LIN {X 0,Y 736.323,Z 990.485,A -85,B 0,C 180,E1 33731.391,E2 33731.391} C_VEL
LIN {X 0,Y 736.504,Z 974.64,A -85,B 0,C 180,E1 33729.663,E2 33729.663} C_VEL
LIN {X 0,Y 736.684,Z 957.169,A -85,B 0,C 180,E1 33728,E2 33728} C_VEL
LIN {X 0,Y 736.943,Z 939.859,A -85,B 0,C 180,E1 33726.521,E2 33726.521} C_VEL
LIN {X 0,Y 737.195,Z 919.804,A -85,B 0,C 180,E1 33725.008,E2 33725.008} C_VEL
LIN {X 0,Y 737.439,Z 901.418,A -85,B 0,C 180,E1 33723.767,E2 33723.767} C_VEL
LIN {X 0,Y 737.809,Z 878.245,A -85,B 0,C 180,E1 33722.388,E2 33722.388} C_VEL
LIN {X 0,Y 738.071,Z 858.185,A -85,B 0,C 180,E1 33721.343,E2 33721.343} C_VEL
LIN {X 0,Y 738.362,Z 837.251,A -85,B 0,C 180,E1 33720.378,E2 33720.378} C_VEL
LIN {X 0,Y 738.709,Z 812.608,A -85,B 0,C 180,E1 33719.407,E2 33719.407} C_VEL
LIN {X 0,Y 738.944,Z 791.175,A -85,B 0,C 180,E1 33718.695,E2 33718.695} C_VEL
LIN {X 0,Y 739.147,Z 770.122,A -85,B 0,C 180,E1 33718.104,E2 33718.104} C_VEL
LIN {X 0,Y 739.421,Z 744.677,A -85,B 0,C 180,E1 33717.531,E2 33717.531} C_VEL
LIN {X 0,Y 739.56,Z 720.624,A -85,B 0,C 180,E1 33717.14,E2 33717.14} C_VEL
LIN {X 0,Y 739.828,Z 623.646,A -85,B 0,C 180,E1 33716.024,E2 33716.024} C_VEL
LIN {X 0,Y 740.398,Z 398.303,A -85,B 0,C 180,E1 33713.431,E2 33713.431} C_VEL
LIN {X 0,Y 740.567,Z 293.06,A -85,B 0,C 180,E1 33712.186,E2 33712.186} C_VEL
LIN {X 0,Y 739.192,Z 287.411,A -85,B 0,C 180,E1 33712.014,E2 33712.014} C_VEL
LIN {X 0,Y 739.245,Z 262.741,A -85,B 0,C 180,E1 33710.326,E2 33710.326} C_VEL
LIN {X 0,Y 736.098,Z 254.481,A -85,B 0,C 180,E1 33709.508,E2 33709.508} C_VEL
LIN {X 0,Y 736.036,Z 254.289,A -85,B 0,C 180,E1 33706.505,E2 33706.505} C_VEL
LIN {X 0,Y 736.021,Z 254.293,A -85,B 0,C 180,E1 33704.057,E2 33704.057} C_VEL
LIN {X 0,Y 736.063,Z 254.286,A -85,B 0,C 180,E1 33701.419,E2 33701.419} C_VEL
LIN {X 0,Y 736.038,Z 254.29,A -85,B 0,C 180,E1 33698.387,E2 33698.387} C_VEL
LIN {X 0,Y 736.02,Z 254.291,A -85,B 0,C 180,E1 33695.936,E2 33695.936} C_VEL
LIN {X 0,Y 736.055,Z 254.282,A -85,B 0,C 180,E1 33693.339,E2 33693.339} C_VEL
LIN {X 0,Y 736.049,Z 254.29,A -85,B 0,C 180,E1 33690.354,E2 33690.354} C_VEL
LIN {X 0,Y 736.019,Z 254.287,A -85,B 0,C 180,E1 33687.824,E2 33687.824} C_VEL
LIN {X 0,Y 736.05,Z 254.289,A -85,B 0,C 180,E1 33685.249,E2 33685.249} C_VEL
LIN {X 0,Y 736.045,Z 254.293,A -85,B 0,C 180,E1 33682.188,E2 33682.188} C_VEL
LIN {X 0,Y 736.018,Z 254.29,A -85,B 0,C 180,E1 33679.689,E2 33679.689} C_VEL
LIN {X 0,Y 736.047,Z 254.288,A -85,B 0,C 180,E1 33677.145,E2 33677.145} C_VEL
LIN {X 0,Y 736.047,Z 254.292,A -85,B 0,C 180,E1 33674.073,E2 33674.073} C_VEL
LIN {X 0,Y 736.019,Z 254.29,A -85,B 0,C 180,E1 33671.52,E2 33671.52} C_VEL
LIN {X 0,Y 736.058,Z 254.288,A -85,B 0,C 180,E1 33668.909,E2 33668.909} C_VEL
LIN {X 0,Y 736.045,Z 254.292,A -85,B 0,C 180,E1 33665.926,E2 33665.926} C_VEL
LIN {X 0,Y 736.018,Z 254.29,A -85,B 0,C 180,E1 33663.427,E2 33663.427} C_VEL
LIN {X 0,Y 736.04,Z 254.289,A -85,B 0,C 180,E1 33660.934,E2 33660.934} C_VEL
LIN {X 0,Y 736.057,Z 254.293,A -85,B 0,C 180,E1 33657.898,E2 33657.898} C_VEL
LIN {X 0,Y 736.018,Z 254.289,A -85,B 0,C 180,E1 33655.325,E2 33655.325} C_VEL
LIN {X 0,Y 736.037,Z 254.289,A -85,B 0,C 180,E1 33652.82,E2 33652.82} C_VEL
LIN {X 0,Y 736.066,Z 254.294,A -85,B 0,C 180,E1 33649.828,E2 33649.828} C_VEL
LIN {X 0,Y 736.017,Z 254.291,A -85,B 0,C 180,E1 33649.201,E2 33649.201} C_VEL
LIN {X 0,Y 735.014,Z 254.419,A -85,B 0,C 180,E1 33648.601,E2 33648.601} C_VEL
LIN {X 0,Y 728.702,Z 255.201,A -85,B 0,C 180,E1 33646.965,E2 33646.965} C_VEL
LIN {X 0,Y 728.126,Z 255.274,A -85,B 0,C 180,E1 33646.485,E2 33646.485} C_VEL
LIN {X 0,Y 728.097,Z 255.278,A -85,B 0,C 180,E1 33643.485,E2 33643.485} C_VEL
LIN {X 0,Y 728.079,Z 255.28,A -85,B 0,C 180,E1 33641.005,E2 33641.005} C_VEL
LIN {X 0,Y 728.121,Z 255.275,A -85,B 0,C 180,E1 33638.385,E2 33638.385} C_VEL
LIN {X 0,Y 728.1,Z 255.276,A -85,B 0,C 180,E1 33635.383,E2 33635.383} C_VEL
LIN {X 0,Y 728.078,Z 255.271,A -85,B 0,C 180,E1 33632.862,E2 33632.862} C_VEL
LIN {X 0,Y 728.117,Z 255.278,A -85,B 0,C 180,E1 33630.281,E2 33630.281} C_VEL
LIN {X 0,Y 728.098,Z 255.27,A -85,B 0,C 180,E1 33627.243,E2 33627.243} C_VEL
LIN {X 0,Y 728.078,Z 255.28,A -85,B 0,C 180,E1 33624.774,E2 33624.774} C_VEL
LIN {X 0,Y 728.106,Z 255.276,A -85,B 0,C 180,E1 33622.231,E2 33622.231} C_VEL
LIN {X 0,Y 728.106,Z 255.281,A -85,B 0,C 180,E1 33619.171,E2 33619.171} C_VEL
LIN {X 0,Y 728.078,Z 255.28,A -85,B 0,C 180,E1 33616.593,E2 33616.593} C_VEL
LIN {X 0,Y 728.121,Z 255.28,A -85,B 0,C 180,E1 33613.98,E2 33613.98} C_VEL
LIN {X 0,Y 728.096,Z 255.277,A -85,B 0,C 180,E1 33610.947,E2 33610.947} C_VEL
LIN {X 0,Y 728.077,Z 255.28,A -85,B 0,C 180,E1 33608.471,E2 33608.471} C_VEL
LIN {X 0,Y 728.174,Z 255.513,A -85,B 0,C 180,E1 33607.228,E2 33607.228} C_VEL
LIN {X 0,Y 732.4,Z 266.408,A -85,B 0,C 180,E1 33606.141,E2 33606.141} C_VEL
LIN {X 0,Y 732.336,Z 278.075,A -85,B 0,C 180,E1 33605.34,E2 33605.34} C_VEL
LIN {X 0,Y 734.39,Z 286.67,A -85,B 0,C 180,E1 33605.1,E2 33605.1} C_VEL
LIN {X 0,Y 733.457,Z 536.818,A -85,B 0,C 180,E1 33602.164,E2 33602.164} C_VEL
LIN {X 0,Y 732.828,Z 710.294,A -85,B 0,C 180,E1 33600.161,E2 33600.161} C_VEL
LIN {X 0,Y 732.643,Z 734.058,A -85,B 0,C 180,E1 33599.773,E2 33599.773} C_VEL
LIN {X 0,Y 732.274,Z 759.946,A -85,B 0,C 180,E1 33599.191,E2 33599.191} C_VEL
LIN {X 0,Y 731.999,Z 780.748,A -85,B 0,C 180,E1 33598.605,E2 33598.605} C_VEL
LIN {X 0,Y 731.681,Z 802.912,A -85,B 0,C 180,E1 33597.863,E2 33597.863} C_VEL
LIN {X 0,Y 731.192,Z 828.846,A -85,B 0,C 180,E1 33596.825,E2 33596.825} C_VEL
LIN {X 0,Y 730.818,Z 849.11,A -85,B 0,C 180,E1 33595.877,E2 33595.877} C_VEL
LIN {X 0,Y 730.44,Z 871.706,A -85,B 0,C 180,E1 33594.677,E2 33594.677} C_VEL
LIN {X 0,Y 729.958,Z 893.15,A -85,B 0,C 180,E1 33593.363,E2 33593.363} C_VEL
LIN {X 0,Y 729.63,Z 912.174,A -85,B 0,C 180,E1 33592.054,E2 33592.054} C_VEL
LIN {X 0,Y 729.24,Z 932.601,A -85,B 0,C 180,E1 33590.465,E2 33590.465} C_VEL
LIN {X 0,Y 728.948,Z 948.78,A -85,B 0,C 180,E1 33589.054,E2 33589.054} C_VEL
LIN {X 0,Y 728.657,Z 967.272,A -85,B 0,C 180,E1 33587.238,E2 33587.238} C_VEL
LIN {X 0,Y 728.462,Z 981.209,A -85,B 0,C 180,E1 33585.688,E2 33585.688} C_VEL
LIN {X 0,Y 728.285,Z 995.564,A -85,B 0,C 180,E1 33583.902,E2 33583.902} C_VEL
LIN {X 0,Y 728.133,Z 1008.414,A -85,B 0,C 180,E1 33582.048,E2 33582.048} C_VEL
LIN {X 0,Y 728.063,Z 1018.17,A -85,B 0,C 180,E1 33580.444,E2 33580.444} C_VEL
LIN {X 0,Y 727.999,Z 1027.486,A -85,B 0,C 180,E1 33578.69,E2 33578.69} C_VEL
LIN {X 0,Y 727.93,Z 1036.565,A -85,B 0,C 180,E1 33576.626,E2 33576.626} C_VEL
LIN {X 0,Y 727.926,Z 1042.525,A -85,B 0,C 180,E1 33574.964,E2 33574.964} C_VEL
LIN {X 0,Y 727.917,Z 1047.127,A -85,B 0,C 180,E1 33573.386,E2 33573.386} C_VEL
LIN {X 0,Y 727.895,Z 1051.021,A -85,B 0,C 180,E1 33571.653,E2 33571.653} C_VEL
LIN {X 0,Y 727.915,Z 1054.124,A -85,B 0,C 180,E1 33569.528,E2 33569.528} C_VEL
LIN {X 0,Y 727.898,Z 1055.29,A -85,B 0,C 180,E1 33567.717,E2 33567.717} C_VEL
LIN {X 0,Y 727.906,Z 1055.253,A -85,B 0,C 180,E1 33566.062,E2 33566.062} C_VEL
LIN {X 0,Y 727.915,Z 1053.741,A -85,B 0,C 180,E1 33563.998,E2 33563.998} C_VEL
LIN {X 0,Y 727.903,Z 1050.624,A -85,B 0,C 180,E1 33562.06,E2 33562.06} C_VEL
LIN {X 0,Y 727.919,Z 1046.681,A -85,B 0,C 180,E1 33560.353,E2 33560.353} C_VEL
LIN {X 0,Y 727.922,Z 1041.132,A -85,B 0,C 180,E1 33558.511,E2 33558.511} C_VEL
LIN {X 0,Y 727.968,Z 1033.315,A -85,B 0,C 180,E1 33556.497,E2 33556.497} C_VEL
LIN {X 0,Y 728.01,Z 1025.304,A -85,B 0,C 180,E1 33554.792,E2 33554.792} C_VEL
LIN {X 0,Y 728.07,Z 1016.391,A -85,B 0,C 180,E1 33553.156,E2 33553.156} C_VEL
LIN {X 0,Y 728.192,Z 1003.884,A -85,B 0,C 180,E1 33551.175,E2 33551.175} C_VEL
LIN {X 0,Y 728.339,Z 991.104,A -85,B 0,C 180,E1 33549.436,E2 33549.436} C_VEL
LIN {X 0,Y 728.522,Z 977.09,A -85,B 0,C 180,E1 33547.74,E2 33547.74} C_VEL
LIN {X 0,Y 728.764,Z 960.225,A -85,B 0,C 180,E1 33545.953,E2 33545.953} C_VEL
LIN {X 0,Y 729.023,Z 944.707,A -85,B 0,C 180,E1 33544.486,E2 33544.486} C_VEL
LIN {X 0,Y 729.396,Z 923.992,A -85,B 0,C 180,E1 33542.751,E2 33542.751} C_VEL
LIN {X 0,Y 729.722,Z 906.229,A -85,B 0,C 180,E1 33541.432,E2 33541.432} C_VEL
LIN {X 0,Y 730.18,Z 884.008,A -85,B 0,C 180,E1 33539.967,E2 33539.967} C_VEL
LIN {X 0,Y 730.522,Z 864.046,A -85,B 0,C 180,E1 33538.811,E2 33538.811} C_VEL
LIN {X 0,Y 730.942,Z 843.542,A -85,B 0,C 180,E1 33537.758,E2 33537.758} C_VEL
LIN {X 0,Y 731.406,Z 818.409,A -85,B 0,C 180,E1 33536.646,E2 33536.646} C_VEL
LIN {X 0,Y 731.725,Z 797.529,A -85,B 0,C 180,E1 33535.856,E2 33535.856} C_VEL
LIN {X 0,Y 732.078,Z 775.308,A -85,B 0,C 180,E1 33535.139,E2 33535.139} C_VEL
LIN {X 0,Y 732.452,Z 749.2,A -85,B 0,C 180,E1 33534.46,E2 33534.46} C_VEL
LIN {X 0,Y 732.673,Z 727.248,A -85,B 0,C 180,E1 33534.016,E2 33534.016} C_VEL
LIN {X 0,Y 732.842,Z 706.664,A -85,B 0,C 180,E1 33533.701,E2 33533.701} C_VEL
LIN {X 0,Y 733.756,Z 454.635,A -85,B 0,C 180,E1 33530.792,E2 33530.792} C_VEL
LIN {X 0,Y 734.238,Z 285.309,A -85,B 0,C 180,E1 33528.784,E2 33528.784} C_VEL
LIN {X 0,Y 732.302,Z 277.803,A -85,B 0,C 180,E1 33528.557,E2 33528.557} C_VEL
LIN {X 0,Y 732.281,Z 266.077,A -85,B 0,C 180,E1 33527.738,E2 33527.738} C_VEL
LIN {X 0,Y 728.187,Z 255.602,A -85,B 0,C 180,E1 33526.699,E2 33526.699} C_VEL
LIN {X 0,Y 728.128,Z 255.249,A -85,B 0,C 180,E1 33526.094,E2 33526.094} C_VEL
LIN {X 0,Y 728.079,Z 255.278,A -85,B 0,C 180,E1 33523.475,E2 33523.475} C_VEL
LIN {X 0,Y 728.096,Z 255.285,A -85,B 0,C 180,E1 33520.948,E2 33520.948} C_VEL
LIN {X 0,Y 728.132,Z 255.273,A -85,B 0,C 180,E1 33517.967,E2 33517.967} C_VEL
LIN {X 0,Y 728.08,Z 255.281,A -85,B 0,C 180,E1 33515.322,E2 33515.322} C_VEL
LIN {X 0,Y 728.095,Z 255.281,A -85,B 0,C 180,E1 33512.812,E2 33512.812} C_VEL
LIN {X 0,Y 728.127,Z 255.277,A -85,B 0,C 180,E1 33509.787,E2 33509.787} C_VEL
LIN {X 0,Y 728.079,Z 255.279,A -85,B 0,C 180,E1 33507.138,E2 33507.138} C_VEL
LIN {X 0,Y 728.103,Z 255.275,A -85,B 0,C 180,E1 33504.589,E2 33504.589} C_VEL
LIN {X 0,Y 728.109,Z 255.274,A -85,B 0,C 180,E1 33501.51,E2 33501.51} C_VEL
LIN {X 0,Y 728.079,Z 255.274,A -85,B 0,C 180,E1 33498.995,E2 33498.995} C_VEL
LIN {X 0,Y 728.107,Z 255.283,A -85,B 0,C 180,E1 33496.433,E2 33496.433} C_VEL
LIN {X 0,Y 728.103,Z 255.27,A -85,B 0,C 180,E1 33493.339,E2 33493.339} C_VEL
LIN {X 0,Y 728.08,Z 255.28,A -85,B 0,C 180,E1 33490.845,E2 33490.845} C_VEL
LIN {X 0,Y 728.108,Z 255.28,A -85,B 0,C 180,E1 33488.291,E2 33488.291} C_VEL
LIN {X 0,Y 728.104,Z 255.276,A -85,B 0,C 180,E1 33485.2,E2 33485.2} C_VEL
LIN {X 0,Y 728.079,Z 255.28,A -85,B 0,C 180,E1 33482.676,E2 33482.676} C_VEL
LIN {X 0,Y 728.117,Z 255.274,A -85,B 0,C 180,E1 33480.079,E2 33480.079} C_VEL
LIN {X 0,Y 728.099,Z 255.279,A -85,B 0,C 180,E1 33477.009,E2 33477.009} C_VEL
LIN {X 0,Y 728.08,Z 255.277,A -85,B 0,C 180,E1 33474.483,E2 33474.483} C_VEL
LIN {X 0,Y 728.14,Z 255.272,A -85,B 0,C 180,E1 33471.789,E2 33471.789} C_VEL
LIN {X 0,Y 728.095,Z 255.277,A -85,B 0,C 180,E1 33468.835,E2 33468.835} C_VEL
LIN {X 0,Y 728.08,Z 255.27,A -85,B 0,C 180,E1 33466.337,E2 33466.337} C_VEL
LIN {X 0,Y 728.141,Z 255.28,A -85,B 0,C 180,E1 33463.65,E2 33463.65} C_VEL
LIN {X 0,Y 728.094,Z 255.271,A -85,B 0,C 180,E1 33460.673,E2 33460.673} C_VEL
LIN {X 0,Y 728.082,Z 255.277,A -85,B 0,C 180,E1 33458.18,E2 33458.18} C_VEL
LIN {X 0,Y 728.145,Z 255.283,A -85,B 0,C 180,E1 33455.499,E2 33455.499} C_VEL
LIN {X 0,Y 728.093,Z 255.278,A -85,B 0,C 180,E1 33452.517,E2 33452.517} C_VEL
LIN {X 0,Y 728.082,Z 255.281,A -85,B 0,C 180,E1 33450.061,E2 33450.061} C_VEL
LIN {X 0,Y 728.147,Z 255.271,A -85,B 0,C 180,E1 33447.327,E2 33447.327} C_VEL
LIN {X 0,Y 728.093,Z 255.28,A -85,B 0,C 180,E1 33444.389,E2 33444.389} C_VEL
LIN {X 0,Y 728.083,Z 255.271,A -85,B 0,C 180,E1 33441.897,E2 33441.897} C_VEL
LIN {X 0,Y 728.154,Z 255.282,A -85,B 0,C 180,E1 33439.167,E2 33439.167} C_VEL
LIN {X 0,Y 728.093,Z 255.28,A -85,B 0,C 180,E1 33436.249,E2 33436.249} C_VEL
LIN {X 0,Y 728.082,Z 255.276,A -85,B 0,C 180,E1 33433.749,E2 33433.749} C_VEL
LIN {X 0,Y 728.193,Z 255.483,A -85,B 0,C 180,E1 33430.95,E2 33430.95} C_VEL
LIN {X 0,Y 732.603,Z 267.238,A -85,B 0,C 180,E1 33429.788,E2 33429.788} C_VEL
LIN {X 0,Y 732.432,Z 288.096,A -85,B 0,C 180,E1 33428.376,E2 33428.376} C_VEL
LIN {X 0,Y 734.386,Z 296.446,A -85,B 0,C 180,E1 33428.148,E2 33428.148} C_VEL
LIN {X 0,Y 733.461,Z 545.298,A -85,B 0,C 180,E1 33425.227,E2 33425.227} C_VEL
LIN {X 0,Y 732.829,Z 720.19,A -85,B 0,C 180,E1 33423.207,E2 33423.207} C_VEL
LIN {X 0,Y 732.646,Z 743.539,A -85,B 0,C 180,E1 33422.827,E2 33422.827} C_VEL
LIN {X 0,Y 732.276,Z 769.69,A -85,B 0,C 180,E1 33422.243,E2 33422.243} C_VEL
LIN {X 0,Y 731.996,Z 791.176,A -85,B 0,C 180,E1 33421.637,E2 33421.637} C_VEL
LIN {X 0,Y 731.671,Z 814.379,A -85,B 0,C 180,E1 33420.856,E2 33420.856} C_VEL
LIN {X 0,Y 731.183,Z 839.24,A -85,B 0,C 180,E1 33419.852,E2 33419.852} C_VEL
LIN {X 0,Y 730.81,Z 859.997,A -85,B 0,C 180,E1 33418.878,E2 33418.878} C_VEL
LIN {X 0,Y 730.41,Z 882.93,A -85,B 0,C 180,E1 33417.65,E2 33417.65} C_VEL
LIN {X 0,Y 729.949,Z 903.562,A -85,B 0,C 180,E1 33416.381,E2 33416.381} C_VEL
LIN {X 0,Y 729.623,Z 922.826,A -85,B 0,C 180,E1 33415.053,E2 33415.053} C_VEL
LIN {X 0,Y 729.242,Z 942.535,A -85,B 0,C 180,E1 33413.516,E2 33413.516} C_VEL
LIN {X 0,Y 728.949,Z 959.029,A -85,B 0,C 180,E1 33412.076,E2 33412.076} C_VEL
LIN {X 0,Y 728.644,Z 977.756,A -85,B 0,C 180,E1 33410.231,E2 33410.231} C_VEL
LIN {X 0,Y 728.462,Z 991.327,A -85,B 0,C 180,E1 33408.719,E2 33408.719} C_VEL
LIN {X 0,Y 728.284,Z 1005.76,A -85,B 0,C 180,E1 33406.922,E2 33406.922} C_VEL
LIN {X 0,Y 728.127,Z 1018.734,A -85,B 0,C 180,E1 33405.043,E2 33405.043} C_VEL
LIN {X 0,Y 728.063,Z 1028.1,A -85,B 0,C 180,E1 33403.501,E2 33403.501} C_VEL
LIN {X 0,Y 727.993,Z 1037.107,A -85,B 0,C 180,E1 33401.809,E2 33401.809} C_VEL
LIN {X 0,Y 727.93,Z 1046.35,A -85,B 0,C 180,E1 33399.727,E2 33399.727} C_VEL
LIN {X 0,Y 727.921,Z 1052.637,A -85,B 0,C 180,E1 33397.975,E2 33397.975} C_VEL
LIN {X 0,Y 727.92,Z 1057.239,A -85,B 0,C 180,E1 33396.388,E2 33396.388} C_VEL
LIN {X 0,Y 727.893,Z 1061.28,A -85,B 0,C 180,E1 33394.57,E2 33394.57} C_VEL
LIN {X 0,Y 727.905,Z 1064.236,A -85,B 0,C 180,E1 33392.441,E2 33392.441} C_VEL
LIN {X 0,Y 727.895,Z 1065.305,A -85,B 0,C 180,E1 33390.708,E2 33390.708} C_VEL
LIN {X 0,Y 727.911,Z 1065.239,A -85,B 0,C 180,E1 33389.056,E2 33389.056} C_VEL
LIN {X 0,Y 727.913,Z 1063.578,A -85,B 0,C 180,E1 33386.929,E2 33386.929} C_VEL
LIN {X 0,Y 727.902,Z 1060.643,A -85,B 0,C 180,E1 33385.114,E2 33385.114} C_VEL
LIN {X 0,Y 727.921,Z 1056.826,A -85,B 0,C 180,E1 33383.454,E2 33383.454} C_VEL
LIN {X 0,Y 727.927,Z 1051.616,A -85,B 0,C 180,E1 33381.707,E2 33381.707} C_VEL
LIN {X 0,Y 727.968,Z 1043.37,A -85,B 0,C 180,E1 33379.554,E2 33379.554} C_VEL
LIN {X 0,Y 728.006,Z 1035.472,A -85,B 0,C 180,E1 33377.87,E2 33377.87} C_VEL
LIN {X 0,Y 728.066,Z 1026.709,A -85,B 0,C 180,E1 33376.256,E2 33376.256} C_VEL
LIN {X 0,Y 728.19,Z 1014.488,A -85,B 0,C 180,E1 33374.306,E2 33374.306} C_VEL
LIN {X 0,Y 728.328,Z 1001.888,A -85,B 0,C 180,E1 33372.581,E2 33372.581} C_VEL
LIN {X 0,Y 728.481,Z 989.069,A -85,B 0,C 180,E1 33371.017,E2 33371.017} C_VEL
LIN {X 0,Y 728.758,Z 972.119,A -85,B 0,C 180,E1 33369.185,E2 33369.185} C_VEL
LIN {X 0,Y 728.981,Z 956.24,A -85,B 0,C 180,E1 33367.67,E2 33367.67} C_VEL
LIN {X 0,Y 729.362,Z 938.18,A -85,B 0,C 180,E1 33366.121,E2 33366.121} C_VEL
LIN {X 0,Y 729.667,Z 918.597,A -85,B 0,C 180,E1 33364.645,E2 33364.645} C_VEL
LIN {X 0,Y 730.065,Z 899.426,A -85,B 0,C 180,E1 33363.35,E2 33363.35} C_VEL
LIN {X 0,Y 730.492,Z 876.503,A -85,B 0,C 180,E1 33361.991,E2 33361.991} C_VEL
LIN {X 0,Y 730.857,Z 856.409,A -85,B 0,C 180,E1 33360.943,E2 33360.943} C_VEL
LIN {X 0,Y 731.357,Z 833.218,A -85,B 0,C 180,E1 33359.884,E2 33359.884} C_VEL
LIN {X 0,Y 731.711,Z 809.195,A -85,B 0,C 180,E1 33358.96,E2 33358.96} C_VEL
LIN {X 0,Y 732.031,Z 787.512,A -85,B 0,C 180,E1 33358.25,E2 33358.25} C_VEL
LIN {X 0,Y 732.441,Z 761.161,A -85,B 0,C 180,E1 33357.548,E2 33357.548} C_VEL
LIN {X 0,Y 732.67,Z 738.074,A -85,B 0,C 180,E1 33357.076,E2 33357.076} C_VEL
LIN {X 0,Y 732.84,Z 717.643,A -85,B 0,C 180,E1 33356.759,E2 33356.759} C_VEL
LIN {X 0,Y 733.755,Z 463.665,A -85,B 0,C 180,E1 33353.826,E2 33353.826} C_VEL
LIN {X 0,Y 734.262,Z 295.156,A -85,B 0,C 180,E1 33351.829,E2 33351.829} C_VEL
LIN {X 0,Y 732.333,Z 287.206,A -85,B 0,C 180,E1 33351.582,E2 33351.582} C_VEL
LIN {X 0,Y 732.518,Z 266.564,A -85,B 0,C 180,E1 33350.158,E2 33350.158} C_VEL
LIN {X 0,Y 728.191,Z 255.47,A -85,B 0,C 180,E1 33349.047,E2 33349.047} C_VEL
LIN {X 0,Y 728.082,Z 255.276,A -85,B 0,C 180,E1 33346.251,E2 33346.251} C_VEL
LIN {X 0,Y 728.094,Z 255.281,A -85,B 0,C 180,E1 33343.751,E2 33343.751} C_VEL
LIN {X 0,Y 728.152,Z 255.284,A -85,B 0,C 180,E1 33340.817,E2 33340.817} C_VEL
LIN {X 0,Y 728.081,Z 255.277,A -85,B 0,C 180,E1 33338.07,E2 33338.07} C_VEL
LIN {X 0,Y 728.094,Z 255.279,A -85,B 0,C 180,E1 33335.611,E2 33335.611} C_VEL
LIN {X 0,Y 728.147,Z 255.279,A -85,B 0,C 180,E1 33332.661,E2 33332.661} C_VEL
LIN {X 0,Y 728.082,Z 255.277,A -85,B 0,C 180,E1 33329.939,E2 33329.939} C_VEL
LIN {X 0,Y 728.093,Z 255.274,A -85,B 0,C 180,E1 33327.48,E2 33327.48} C_VEL
LIN {X 0,Y 728.144,Z 255.28,A -85,B 0,C 180,E1 33324.501,E2 33324.501} C_VEL
LIN {X 0,Y 728.082,Z 255.281,A -85,B 0,C 180,E1 33321.82,E2 33321.82} C_VEL
LIN {X 0,Y 728.092,Z 255.278,A -85,B 0,C 180,E1 33319.328,E2 33319.328} C_VEL
LIN {X 0,Y 728.141,Z 255.282,A -85,B 0,C 180,E1 33316.35,E2 33316.35} C_VEL
LIN {X 0,Y 728.081,Z 255.279,A -85,B 0,C 180,E1 33313.663,E2 33313.663} C_VEL
LIN {X 0,Y 728.095,Z 255.278,A -85,B 0,C 180,E1 33311.165,E2 33311.165} C_VEL
LIN {X 0,Y 728.14,Z 255.282,A -85,B 0,C 180,E1 33308.211,E2 33308.211} C_VEL
LIN {X 0,Y 728.082,Z 255.28,A -85,B 0,C 180,E1 33305.596,E2 33305.596} C_VEL
LIN {X 0,Y 728.087,Z 255.278,A -85,B 0,C 180,E1 33303.149,E2 33303.149} C_VEL
LIN {X 0,Y 728.159,Z 255.279,A -85,B 0,C 180,E1 33300.236,E2 33300.236} C_VEL
LIN {X 0,Y 728.082,Z 255.281,A -85,B 0,C 180,E1 33297.481,E2 33297.481} C_VEL
LIN {X 0,Y 728.085,Z 255.276,A -85,B 0,C 180,E1 33295.037,E2 33295.037} C_VEL
LIN {X 0,Y 728.163,Z 255.281,A -85,B 0,C 180,E1 33292.187,E2 33292.187} C_VEL
LIN {X 0,Y 728.085,Z 255.281,A -85,B 0,C 180,E1 33289.396,E2 33289.396} C_VEL
LIN {X 0,Y 728.085,Z 255.275,A -85,B 0,C 180,E1 33286.903,E2 33286.903} C_VEL
LIN {X 0,Y 728.126,Z 255.274,A -85,B 0,C 180,E1 33286.485,E2 33286.485} C_VEL
LIN {X 0,Y 727.213,Z 255.4,A -85,B 0,C 180,E1 33285.879,E2 33285.879} C_VEL
LIN {X 0,Y 720.673,Z 256.214,A -85,B 0,C 180,E1 33284.139,E2 33284.139} C_VEL
LIN {X 0,Y 720.189,Z 256.267,A -85,B 0,C 180,E1 33283.741,E2 33283.741} C_VEL
LIN {X 0,Y 720.142,Z 256.27,A -85,B 0,C 180,E1 33281.124,E2 33281.124} C_VEL
LIN {X 0,Y 720.16,Z 256.264,A -85,B 0,C 180,E1 33278.583,E2 33278.583} C_VEL
LIN {X 0,Y 720.181,Z 256.264,A -85,B 0,C 180,E1 33275.56,E2 33275.56} C_VEL
LIN {X 0,Y 720.14,Z 256.259,A -85,B 0,C 180,E1 33272.997,E2 33272.997} C_VEL
LIN {X 0,Y 720.153,Z 256.268,A -85,B 0,C 180,E1 33270.522,E2 33270.522} C_VEL
LIN {X 0,Y 720.203,Z 256.256,A -85,B 0,C 180,E1 33267.576,E2 33267.576} C_VEL
LIN {X 0,Y 720.14,Z 256.27,A -85,B 0,C 180,E1 33264.865,E2 33264.865} C_VEL
LIN {X 0,Y 720.156,Z 256.266,A -85,B 0,C 180,E1 33262.344,E2 33262.344} C_VEL
LIN {X 0,Y 720.193,Z 256.268,A -85,B 0,C 180,E1 33259.372,E2 33259.372} C_VEL
LIN {X 0,Y 720.139,Z 256.269,A -85,B 0,C 180,E1 33256.682,E2 33256.682} C_VEL
LIN {X 0,Y 720.165,Z 256.27,A -85,B 0,C 180,E1 33254.125,E2 33254.125} C_VEL
LIN {X 0,Y 720.167,Z 256.264,A -85,B 0,C 180,E1 33251.05,E2 33251.05} C_VEL
LIN {X 0,Y 720.139,Z 256.27,A -85,B 0,C 180,E1 33248.566,E2 33248.566} C_VEL
LIN {X 0,Y 720.245,Z 256.505,A -85,B 0,C 180,E1 33247.691,E2 33247.691} C_VEL
LIN {X 0,Y 725.531,Z 270.252,A -85,B 0,C 180,E1 33246.306,E2 33246.306} C_VEL
LIN {X 0,Y 725.449,Z 277.719,A -85,B 0,C 180,E1 33245.786,E2 33245.786} C_VEL
LIN {X 0,Y 728.079,Z 288.669,A -85,B 0,C 180,E1 33245.466,E2 33245.466} C_VEL
LIN {X 0,Y 726.907,Z 538.233,A -85,B 0,C 180,E1 33242.513,E2 33242.513} C_VEL
LIN {X 0,Y 726.122,Z 710.327,A -85,B 0,C 180,E1 33240.507,E2 33240.507} C_VEL
LIN {X 0,Y 725.882,Z 734.884,A -85,B 0,C 180,E1 33240.103,E2 33240.103} C_VEL
LIN {X 0,Y 725.421,Z 760.555,A -85,B 0,C 180,E1 33239.516,E2 33239.516} C_VEL
LIN {X 0,Y 725.066,Z 782.126,A -85,B 0,C 180,E1 33238.9,E2 33238.9} C_VEL
LIN {X 0,Y 724.64,Z 806.426,A -85,B 0,C 180,E1 33238.068,E2 33238.068} C_VEL
LIN {X 0,Y 724.063,Z 829.695,A -85,B 0,C 180,E1 33237.11,E2 33237.11} C_VEL
LIN {X 0,Y 723.584,Z 849.875,A -85,B 0,C 180,E1 33236.156,E2 33236.156} C_VEL
LIN {X 0,Y 723.065,Z 873.342,A -85,B 0,C 180,E1 33234.885,E2 33234.885} C_VEL
LIN {X 0,Y 722.525,Z 893.503,A -85,B 0,C 180,E1 33233.632,E2 33233.632} C_VEL
LIN {X 0,Y 722.082,Z 913.289,A -85,B 0,C 180,E1 33232.254,E2 33232.254} C_VEL
LIN {X 0,Y 721.611,Z 933.039,A -85,B 0,C 180,E1 33230.691,E2 33230.691} C_VEL
LIN {X 0,Y 721.226,Z 949.429,A -85,B 0,C 180,E1 33229.243,E2 33229.243} C_VEL
LIN {X 0,Y 720.857,Z 968.029,A -85,B 0,C 180,E1 33227.385,E2 33227.385} C_VEL
LIN {X 0,Y 720.606,Z 981.518,A -85,B 0,C 180,E1 33225.864,E2 33225.864} C_VEL
LIN {X 0,Y 720.387,Z 996.117,A -85,B 0,C 180,E1 33224.02,E2 33224.02} C_VEL
LIN {X 0,Y 720.21,Z 1008.64,A -85,B 0,C 180,E1 33222.182,E2 33222.182} C_VEL
LIN {X 0,Y 720.101,Z 1018.43,A -85,B 0,C 180,E1 33220.551,E2 33220.551} C_VEL
LIN {X 0,Y 720.023,Z 1028.06,A -85,B 0,C 180,E1 33218.706,E2 33218.706} C_VEL
LIN {X 0,Y 719.942,Z 1036.696,A -85,B 0,C 180,E1 33216.699,E2 33216.699} C_VEL
LIN {X 0,Y 719.933,Z 1042.634,A -85,B 0,C 180,E1 33215.02,E2 33215.02} C_VEL
LIN {X 0,Y 719.918,Z 1047.421,A -85,B 0,C 180,E1 33213.344,E2 33213.344} C_VEL
LIN {X 0,Y 719.897,Z 1051.724,A -85,B 0,C 180,E1 33211.353,E2 33211.353} C_VEL
LIN {X 0,Y 719.902,Z 1054.287,A -85,B 0,C 180,E1 33209.363,E2 33209.363} C_VEL
LIN {X 0,Y 719.897,Z 1055.3,A -85,B 0,C 180,E1 33207.692,E2 33207.692} C_VEL
LIN {X 0,Y 719.914,Z 1055.221,A -85,B 0,C 180,E1 33205.938,E2 33205.938} C_VEL
LIN {X 0,Y 719.911,Z 1053.48,A -85,B 0,C 180,E1 33203.781,E2 33203.781} C_VEL
LIN {X 0,Y 719.914,Z 1050.486,A -85,B 0,C 180,E1 33201.936,E2 33201.936} C_VEL
LIN {X 0,Y 719.92,Z 1046.592,A -85,B 0,C 180,E1 33200.245,E2 33200.245} C_VEL
LIN {X 0,Y 719.928,Z 1040.708,A -85,B 0,C 180,E1 33198.283,E2 33198.283} C_VEL
LIN {X 0,Y 719.976,Z 1032.8,A -85,B 0,C 180,E1 33196.262,E2 33196.262} C_VEL
LIN {X 0,Y 720.042,Z 1025.126,A -85,B 0,C 180,E1 33194.619,E2 33194.619} C_VEL
LIN {X 0,Y 720.132,Z 1016.188,A -85,B 0,C 180,E1 33192.964,E2 33192.964} C_VEL
LIN {X 0,Y 720.273,Z 1003.627,A -85,B 0,C 180,E1 33190.96,E2 33190.96} C_VEL
LIN {X 0,Y 720.453,Z 991.383,A -85,B 0,C 180,E1 33189.274,E2 33189.274} C_VEL
LIN {X 0,Y 720.672,Z 978.219,A -85,B 0,C 180,E1 33187.657,E2 33187.657} C_VEL
LIN {X 0,Y 720.991,Z 960.711,A -85,B 0,C 180,E1 33185.764,E2 33185.764} C_VEL
LIN {X 0,Y 721.332,Z 945.28,A -85,B 0,C 180,E1 33184.287,E2 33184.287} C_VEL
LIN {X 0,Y 721.776,Z 925.758,A -85,B 0,C 180,E1 33182.618,E2 33182.618} C_VEL
LIN {X 0,Y 722.193,Z 907.48,A -85,B 0,C 180,E1 33181.237,E2 33181.237} C_VEL
LIN {X 0,Y 722.757,Z 886.34,A -85,B 0,C 180,E1 33179.81,E2 33179.81} C_VEL
LIN {X 0,Y 723.218,Z 864.818,A -85,B 0,C 180,E1 33178.544,E2 33178.544} C_VEL
LIN {X 0,Y 723.734,Z 844.581,A -85,B 0,C 180,E1 33177.491,E2 33177.491} C_VEL
LIN {X 0,Y 724.313,Z 820.131,A -85,B 0,C 180,E1 33176.388,E2 33176.388} C_VEL
LIN {X 0,Y 724.736,Z 797.705,A -85,B 0,C 180,E1 33175.528,E2 33175.528} C_VEL
LIN {X 0,Y 725.193,Z 775.515,A -85,B 0,C 180,E1 33174.807,E2 33174.807} C_VEL
LIN {X 0,Y 725.649,Z 749.509,A -85,B 0,C 180,E1 33174.124,E2 33174.124} C_VEL
LIN {X 0,Y 725.927,Z 727.167,A -85,B 0,C 180,E1 33173.669,E2 33173.669} C_VEL
LIN {X 0,Y 726.141,Z 706.112,A -85,B 0,C 180,E1 33173.346,E2 33173.346} C_VEL
LIN {X 0,Y 727.279,Z 456.937,A -85,B 0,C 180,E1 33170.446,E2 33170.446} C_VEL
LIN {X 0,Y 727.934,Z 287.281,A -85,B 0,C 180,E1 33168.417,E2 33168.417} C_VEL
LIN {X 0,Y 725.457,Z 277.785,A -85,B 0,C 180,E1 33168.127,E2 33168.127} C_VEL
LIN {X 0,Y 725.463,Z 269.806,A -85,B 0,C 180,E1 33167.567,E2 33167.567} C_VEL
LIN {X 0,Y 720.24,Z 256.467,A -85,B 0,C 180,E1 33166.212,E2 33166.212} C_VEL
LIN {X 0,Y 720.143,Z 256.265,A -85,B 0,C 180,E1 33163.526,E2 33163.526} C_VEL
LIN {X 0,Y 720.15,Z 256.274,A -85,B 0,C 180,E1 33161.052,E2 33161.052} C_VEL
LIN {X 0,Y 720.216,Z 256.261,A -85,B 0,C 180,E1 33158.156,E2 33158.156} C_VEL
LIN {X 0,Y 720.143,Z 256.27,A -85,B 0,C 180,E1 33155.38,E2 33155.38} C_VEL
LIN {X 0,Y 720.153,Z 256.27,A -85,B 0,C 180,E1 33152.86,E2 33152.86} C_VEL
LIN {X 0,Y 720.204,Z 256.266,A -85,B 0,C 180,E1 33149.895,E2 33149.895} C_VEL
LIN {X 0,Y 720.141,Z 256.267,A -85,B 0,C 180,E1 33147.181,E2 33147.181} C_VEL
LIN {X 0,Y 720.153,Z 256.263,A -85,B 0,C 180,E1 33144.704,E2 33144.704} C_VEL
LIN {X 0,Y 720.204,Z 256.261,A -85,B 0,C 180,E1 33141.752,E2 33141.752} C_VEL
LIN {X 0,Y 720.141,Z 256.262,A -85,B 0,C 180,E1 33139.044,E2 33139.044} C_VEL
LIN {X 0,Y 720.158,Z 256.271,A -85,B 0,C 180,E1 33136.537,E2 33136.537} C_VEL
LIN {X 0,Y 720.182,Z 256.257,A -85,B 0,C 180,E1 33133.488,E2 33133.488} C_VEL
LIN {X 0,Y 720.141,Z 256.269,A -85,B 0,C 180,E1 33130.885,E2 33130.885} C_VEL
LIN {X 0,Y 720.168,Z 256.269,A -85,B 0,C 180,E1 33128.302,E2 33128.302} C_VEL
LIN {X 0,Y 720.164,Z 256.265,A -85,B 0,C 180,E1 33125.178,E2 33125.178} C_VEL
LIN {X 0,Y 720.141,Z 256.269,A -85,B 0,C 180,E1 33122.626,E2 33122.626} C_VEL
LIN {X 0,Y 720.2,Z 256.258,A -85,B 0,C 180,E1 33119.92,E2 33119.92} C_VEL
LIN {X 0,Y 720.157,Z 256.268,A -85,B 0,C 180,E1 33116.976,E2 33116.976} C_VEL
LIN {X 0,Y 720.141,Z 256.266,A -85,B 0,C 180,E1 33114.502,E2 33114.502} C_VEL
LIN {X 0,Y 720.19,Z 256.258,A -85,B 0,C 180,E1 33111.85,E2 33111.85} C_VEL
LIN {X 0,Y 720.16,Z 256.266,A -85,B 0,C 180,E1 33108.873,E2 33108.873} C_VEL
LIN {X 0,Y 720.141,Z 256.257,A -85,B 0,C 180,E1 33106.347,E2 33106.347} C_VEL
LIN {X 0,Y 720.204,Z 256.268,A -85,B 0,C 180,E1 33103.63,E2 33103.63} C_VEL
LIN {X 0,Y 720.158,Z 256.259,A -85,B 0,C 180,E1 33100.704,E2 33100.704} C_VEL
LIN {X 0,Y 720.142,Z 256.265,A -85,B 0,C 180,E1 33098.24,E2 33098.24} C_VEL
LIN {X 0,Y 720.196,Z 256.273,A -85,B 0,C 180,E1 33095.56,E2 33095.56} C_VEL
LIN {X 0,Y 720.157,Z 256.267,A -85,B 0,C 180,E1 33092.551,E2 33092.551} C_VEL
LIN {X 0,Y 720.144,Z 256.271,A -85,B 0,C 180,E1 33090.042,E2 33090.042} C_VEL
LIN {X 0,Y 720.214,Z 256.255,A -85,B 0,C 180,E1 33087.28,E2 33087.28} C_VEL
LIN {X 0,Y 720.158,Z 256.269,A -85,B 0,C 180,E1 33084.426,E2 33084.426} C_VEL
LIN {X 0,Y 720.143,Z 256.258,A -85,B 0,C 180,E1 33081.929,E2 33081.929} C_VEL
LIN {X 0,Y 720.215,Z 256.27,A -85,B 0,C 180,E1 33079.163,E2 33079.163} C_VEL
LIN {X 0,Y 720.153,Z 256.27,A -85,B 0,C 180,E1 33076.219,E2 33076.219} C_VEL
LIN {X 0,Y 720.143,Z 256.264,A -85,B 0,C 180,E1 33073.745,E2 33073.745} C_VEL
LIN {X 0,Y 720.192,Z 256.474,A -85,B 0,C 180,E1 33071.434,E2 33071.434} C_VEL
LIN {X 0,Y 725.799,Z 270.471,A -85,B 0,C 180,E1 33070.006,E2 33070.006} C_VEL
LIN {X 0,Y 725.612,Z 288.098,A -85,B 0,C 180,E1 33068.805,E2 33068.805} C_VEL
LIN {X 0,Y 728.077,Z 298.415,A -85,B 0,C 180,E1 33068.515,E2 33068.515} C_VEL
LIN {X 0,Y 726.912,Z 546.785,A -85,B 0,C 180,E1 33065.574,E2 33065.574} C_VEL
LIN {X 0,Y 726.121,Z 720.297,A -85,B 0,C 180,E1 33063.553,E2 33063.553} C_VEL
LIN {X 0,Y 725.884,Z 744.674,A -85,B 0,C 180,E1 33063.152,E2 33063.152} C_VEL
LIN {X 0,Y 725.422,Z 770.447,A -85,B 0,C 180,E1 33062.564,E2 33062.564} C_VEL
LIN {X 0,Y 725.068,Z 791.914,A -85,B 0,C 180,E1 33061.951,E2 33061.951} C_VEL
LIN {X 0,Y 724.64,Z 816.396,A -85,B 0,C 180,E1 33061.114,E2 33061.114} C_VEL
LIN {X 0,Y 724.047,Z 840.237,A -85,B 0,C 180,E1 33060.131,E2 33060.131} C_VEL
LIN {X 0,Y 723.569,Z 860.902,A -85,B 0,C 180,E1 33059.149,E2 33059.149} C_VEL
LIN {X 0,Y 723.012,Z 885.131,A -85,B 0,C 180,E1 33057.823,E2 33057.823} C_VEL
LIN {X 0,Y 722.498,Z 904.433,A -85,B 0,C 180,E1 33056.616,E2 33056.616} C_VEL
LIN {X 0,Y 722.051,Z 925.219,A -85,B 0,C 180,E1 33055.159,E2 33055.159} C_VEL
LIN {X 0,Y 721.58,Z 943.956,A -85,B 0,C 180,E1 33053.659,E2 33053.659} C_VEL
LIN {X 0,Y 721.209,Z 961.347,A -85,B 0,C 180,E1 33052.111,E2 33052.111} C_VEL
LIN {X 0,Y 720.842,Z 978.536,A -85,B 0,C 180,E1 33050.375,E2 33050.375} C_VEL
LIN {X 0,Y 720.605,Z 991.954,A -85,B 0,C 180,E1 33048.857,E2 33048.857} C_VEL
LIN {X 0,Y 720.377,Z 1006.632,A -85,B 0,C 180,E1 33046.992,E2 33046.992} C_VEL
LIN {X 0,Y 720.208,Z 1018.735,A -85,B 0,C 180,E1 33045.212,E2 33045.212} C_VEL
LIN {X 0,Y 720.102,Z 1028.565,A -85,B 0,C 180,E1 33043.572,E2 33043.572} C_VEL
LIN {X 0,Y 720.027,Z 1038.729,A -85,B 0,C 180,E1 33041.616,E2 33041.616} C_VEL
LIN {X 0,Y 719.938,Z 1046.961,A -85,B 0,C 180,E1 33039.675,E2 33039.675} C_VEL
LIN {X 0,Y 719.926,Z 1052.892,A -85,B 0,C 180,E1 33037.983,E2 33037.983} C_VEL
LIN {X 0,Y 719.916,Z 1057.652,A -85,B 0,C 180,E1 33036.299,E2 33036.299} C_VEL
LIN {X 0,Y 719.908,Z 1061.997,A -85,B 0,C 180,E1 33034.222,E2 33034.222} C_VEL
LIN {X 0,Y 719.901,Z 1064.371,A -85,B 0,C 180,E1 33032.308,E2 33032.308} C_VEL
LIN {X 0,Y 719.893,Z 1065.328,A -85,B 0,C 180,E1 33030.637,E2 33030.637} C_VEL
LIN {X 0,Y 719.916,Z 1065.172,A -85,B 0,C 180,E1 33028.806,E2 33028.806} C_VEL
LIN {X 0,Y 719.904,Z 1063.24,A -85,B 0,C 180,E1 33026.656,E2 33026.656} C_VEL
LIN {X 0,Y 719.917,Z 1060.325,A -85,B 0,C 180,E1 33024.9,E2 33024.9} C_VEL
LIN {X 0,Y 719.919,Z 1056.206,A -85,B 0,C 180,E1 33023.14,E2 33023.14} C_VEL
LIN {X 0,Y 719.952,Z 1049.4,A -85,B 0,C 180,E1 33020.971,E2 33020.971} C_VEL
LIN {X 0,Y 719.975,Z 1042.303,A -85,B 0,C 180,E1 33019.194,E2 33019.194} C_VEL
LIN {X 0,Y 720.041,Z 1034.655,A -85,B 0,C 180,E1 33017.57,E2 33017.57} C_VEL
LIN {X 0,Y 720.162,Z 1024.391,A -85,B 0,C 180,E1 33015.692,E2 33015.692} C_VEL
LIN {X 0,Y 720.288,Z 1012.179,A -85,B 0,C 180,E1 33013.798,E2 33013.798} C_VEL
LIN {X 0,Y 720.467,Z 999.996,A -85,B 0,C 180,E1 33012.139,E2 33012.139} C_VEL
LIN {X 0,Y 720.763,Z 984.743,A -85,B 0,C 180,E1 33010.3,E2 33010.3} C_VEL
LIN {X 0,Y 721.006,Z 969.566,A -85,B 0,C 180,E1 33008.695,E2 33008.695} C_VEL
LIN {X 0,Y 721.388,Z 953.45,A -85,B 0,C 180,E1 33007.164,E2 33007.164} C_VEL
LIN {X 0,Y 721.799,Z 933.978,A -85,B 0,C 180,E1 33005.523,E2 33005.523} C_VEL
LIN {X 0,Y 722.232,Z 916.182,A -85,B 0,C 180,E1 33004.189,E2 33004.189} C_VEL
LIN {X 0,Y 722.785,Z 893.865,A -85,B 0,C 180,E1 33002.704,E2 33002.704} C_VEL
LIN {X 0,Y 723.262,Z 873.436,A -85,B 0,C 180,E1 33001.514,E2 33001.514} C_VEL
LIN {X 0,Y 723.82,Z 851.929,A -85,B 0,C 180,E1 33000.406,E2 33000.406} C_VEL
LIN {X 0,Y 724.348,Z 827.242,A -85,B 0,C 180,E1 32999.316,E2 32999.316} C_VEL
LIN {X 0,Y 724.765,Z 806.254,A -85,B 0,C 180,E1 32998.522,E2 32998.522} C_VEL
LIN {X 0,Y 725.322,Z 781.518,A -85,B 0,C 180,E1 32997.733,E2 32997.733} C_VEL
LIN {X 0,Y 725.674,Z 756.594,A -85,B 0,C 180,E1 32997.104,E2 32997.104} C_VEL
LIN {X 0,Y 725.939,Z 735.289,A -85,B 0,C 180,E1 32996.68,E2 32996.68} C_VEL
LIN {X 0,Y 726.175,Z 711.632,A -85,B 0,C 180,E1 32996.33,E2 32996.33} C_VEL
LIN {X 0,Y 727.276,Z 467.522,A -85,B 0,C 180,E1 32993.498,E2 32993.498} C_VEL
LIN {X 0,Y 727.944,Z 297.041,A -85,B 0,C 180,E1 32991.46,E2 32991.46} C_VEL
LIN {X 0,Y 725.524,Z 287.445,A -85,B 0,C 180,E1 32991.167,E2 32991.167} C_VEL
LIN {X 0,Y 725.613,Z 269.968,A -85,B 0,C 180,E1 32989.945,E2 32989.945} C_VEL
LIN {X 0,Y 720.193,Z 256.476,A -85,B 0,C 180,E1 32988.566,E2 32988.566} C_VEL
LIN {X 0,Y 720.142,Z 256.262,A -85,B 0,C 180,E1 32986.034,E2 32986.034} C_VEL
LIN {X 0,Y 720.208,Z 256.262,A -85,B 0,C 180,E1 32983.302,E2 32983.302} C_VEL
LIN {X 0,Y 720.155,Z 256.271,A -85,B 0,C 180,E1 32980.337,E2 32980.337} C_VEL
LIN {X 0,Y 720.145,Z 256.265,A -85,B 0,C 180,E1 32977.812,E2 32977.812} C_VEL
LIN {X 0,Y 720.22,Z 256.265,A -85,B 0,C 180,E1 32974.986,E2 32974.986} C_VEL
LIN {X 0,Y 720.148,Z 256.271,A -85,B 0,C 180,E1 32972.119,E2 32972.119} C_VEL
LIN {X 0,Y 720.146,Z 256.264,A -85,B 0,C 180,E1 32969.623,E2 32969.623} C_VEL
LIN {X 0,Y 720.224,Z 256.263,A -85,B 0,C 180,E1 32966.789,E2 32966.789} C_VEL
LIN {X 0,Y 720.148,Z 256.268,A -85,B 0,C 180,E1 32963.993,E2 32963.993} C_VEL
LIN {X 0,Y 720.146,Z 256.268,A -85,B 0,C 180,E1 32961.503,E2 32961.503} C_VEL
LIN {X 0,Y 720.223,Z 256.266,A -85,B 0,C 180,E1 32958.705,E2 32958.705} C_VEL
LIN {X 0,Y 720.146,Z 256.269,A -85,B 0,C 180,E1 32955.805,E2 32955.805} C_VEL
LIN {X 0,Y 720.148,Z 256.267,A -85,B 0,C 180,E1 32953.326,E2 32953.326} C_VEL
LIN {X 0,Y 720.218,Z 256.272,A -85,B 0,C 180,E1 32950.398,E2 32950.398} C_VEL
LIN {X 0,Y 720.145,Z 256.269,A -85,B 0,C 180,E1 32947.66,E2 32947.66} C_VEL
LIN {X 0,Y 720.149,Z 256.267,A -85,B 0,C 180,E1 32945.178,E2 32945.178} C_VEL
LIN {X 0,Y 720.22,Z 256.27,A -85,B 0,C 180,E1 32942.307,E2 32942.307} C_VEL
LIN {X 0,Y 720.144,Z 256.268,A -85,B 0,C 180,E1 32939.523,E2 32939.523} C_VEL
LIN {X 0,Y 720.148,Z 256.268,A -85,B 0,C 180,E1 32937.055,E2 32937.055} C_VEL
LIN {X 0,Y 720.218,Z 256.27,A -85,B 0,C 180,E1 32934.103,E2 32934.103} C_VEL
LIN {X 0,Y 720.142,Z 256.266,A -85,B 0,C 180,E1 32931.332,E2 32931.332} C_VEL
LIN {X 0,Y 720.151,Z 256.268,A -85,B 0,C 180,E1 32928.872,E2 32928.872} C_VEL
LIN {X 0,Y 720.216,Z 256.27,A -85,B 0,C 180,E1 32925.939,E2 32925.939} C_VEL
LIN {X 0,Y 720.189,Z 256.267,A -85,B 0,C 180,E1 32923.741,E2 32923.741} C_VEL
LIN {X 0,Y 719.144,Z 256.391,A -85,B 0,C 180,E1 32923.128,E2 32923.128} C_VEL
LIN {X 0,Y 712.727,Z 257.199,A -85,B 0,C 180,E1 32921.411,E2 32921.411} C_VEL
LIN {X 0,Y 712.203,Z 257.258,A -85,B 0,C 180,E1 32920.965,E2 32920.965} C_VEL
LIN {X 0,Y 712.264,Z 257.251,A -85,B 0,C 180,E1 32918.247,E2 32918.247} C_VEL
LIN {X 0,Y 712.212,Z 257.251,A -85,B 0,C 180,E1 32915.268,E2 32915.268} C_VEL
LIN {X 0,Y 712.202,Z 257.245,A -85,B 0,C 180,E1 32912.762,E2 32912.762} C_VEL
LIN {X 0,Y 712.287,Z 257.256,A -85,B 0,C 180,E1 32909.924,E2 32909.924} C_VEL
LIN {X 0,Y 712.208,Z 257.242,A -85,B 0,C 180,E1 32907.09,E2 32907.09} C_VEL
LIN {X 0,Y 712.204,Z 257.258,A -85,B 0,C 180,E1 32904.655,E2 32904.655} C_VEL
LIN {X 0,Y 712.276,Z 257.252,A -85,B 0,C 180,E1 32901.854,E2 32901.854} C_VEL
LIN {X 0,Y 712.208,Z 257.258,A -85,B 0,C 180,E1 32898.925,E2 32898.925} C_VEL
LIN {X 0,Y 712.205,Z 257.257,A -85,B 0,C 180,E1 32896.421,E2 32896.421} C_VEL
LIN {X 0,Y 712.285,Z 257.253,A -85,B 0,C 180,E1 32893.571,E2 32893.571} C_VEL
LIN {X 0,Y 712.204,Z 257.252,A -85,B 0,C 180,E1 32890.755,E2 32890.755} C_VEL
LIN {X 0,Y 712.215,Z 257.322,A -85,B 0,C 180,E1 32888.252,E2 32888.252} C_VEL
LIN {X 0,Y 712.336,Z 257.947,A -85,B 0,C 180,E1 32888.111,E2 32888.111} C_VEL
LIN {X 0,Y 718.674,Z 273.783,A -85,B 0,C 180,E1 32886.497,E2 32886.497} C_VEL
LIN {X 0,Y 718.77,Z 278.477,A -85,B 0,C 180,E1 32886.194,E2 32886.194} C_VEL
LIN {X 0,Y 721.8,Z 290.609,A -85,B 0,C 180,E1 32885.84,E2 32885.84} C_VEL
LIN {X 0,Y 720.385,Z 539.475,A -85,B 0,C 180,E1 32882.869,E2 32882.869} C_VEL
LIN {X 0,Y 719.44,Z 710.464,A -85,B 0,C 180,E1 32880.859,E2 32880.859} C_VEL
LIN {X 0,Y 719.143,Z 735.502,A -85,B 0,C 180,E1 32880.442,E2 32880.442} C_VEL
LIN {X 0,Y 718.599,Z 760.953,A -85,B 0,C 180,E1 32879.854,E2 32879.854} C_VEL
LIN {X 0,Y 718.166,Z 782.508,A -85,B 0,C 180,E1 32879.231,E2 32879.231} C_VEL
LIN {X 0,Y 717.62,Z 807.382,A -85,B 0,C 180,E1 32878.368,E2 32878.368} C_VEL
LIN {X 0,Y 716.954,Z 830.543,A -85,B 0,C 180,E1 32877.402,E2 32877.402} C_VEL
LIN {X 0,Y 716.353,Z 851.506,A -85,B 0,C 180,E1 32876.395,E2 32876.395} C_VEL
LIN {X 0,Y 715.67,Z 875.833,A -85,B 0,C 180,E1 32875.045,E2 32875.045} C_VEL
LIN {X 0,Y 715.071,Z 894.943,A -85,B 0,C 180,E1 32873.835,E2 32873.835} C_VEL
LIN {X 0,Y 714.51,Z 915.531,A -85,B 0,C 180,E1 32872.373,E2 32872.373} C_VEL
LIN {X 0,Y 713.954,Z 934.472,A -85,B 0,C 180,E1 32870.838,E2 32870.838} C_VEL
LIN {X 0,Y 713.48,Z 952.311,A -85,B 0,C 180,E1 32869.228,E2 32869.228} C_VEL
LIN {X 0,Y 713.042,Z 969.446,A -85,B 0,C 180,E1 32867.463,E2 32867.463} C_VEL
LIN {X 0,Y 712.746,Z 983.222,A -85,B 0,C 180,E1 32865.876,E2 32865.876} C_VEL
LIN {X 0,Y 712.448,Z 998.405,A -85,B 0,C 180,E1 32863.886,E2 32863.886} C_VEL
LIN {X 0,Y 712.273,Z 1009.381,A -85,B 0,C 180,E1 32862.238,E2 32862.238} C_VEL
LIN {X 0,Y 712.14,Z 1019.489,A -85,B 0,C 180,E1 32860.517,E2 32860.517} C_VEL
LIN {X 0,Y 712.036,Z 1030.068,A -85,B 0,C 180,E1 32858.398,E2 32858.398} C_VEL
LIN {X 0,Y 711.949,Z 1037.432,A -85,B 0,C 180,E1 32856.613,E2 32856.613} C_VEL
LIN {X 0,Y 711.935,Z 1043.251,A -85,B 0,C 180,E1 32854.915,E2 32854.915} C_VEL
LIN {X 0,Y 711.919,Z 1048.537,A -85,B 0,C 180,E1 32852.979,E2 32852.979} C_VEL
LIN {X 0,Y 711.919,Z 1052.473,A -85,B 0,C 180,E1 32850.885,E2 32850.885} C_VEL
LIN {X 0,Y 711.904,Z 1054.45,A -85,B 0,C 180,E1 32849.195,E2 32849.195} C_VEL
LIN {X 0,Y 711.891,Z 1055.376,A -85,B 0,C 180,E1 32847.424,E2 32847.424} C_VEL
LIN {X 0,Y 711.894,Z 1054.961,A -85,B 0,C 180,E1 32845.327,E2 32845.327} C_VEL
LIN {X 0,Y 711.903,Z 1053.092,A -85,B 0,C 180,E1 32843.467,E2 32843.467} C_VEL
LIN {X 0,Y 711.915,Z 1050.258,A -85,B 0,C 180,E1 32841.764,E2 32841.764} C_VEL
LIN {X 0,Y 711.925,Z 1046.086,A -85,B 0,C 180,E1 32839.97,E2 32839.97} C_VEL
LIN {X 0,Y 711.967,Z 1039.15,A -85,B 0,C 180,E1 32837.757,E2 32837.757} C_VEL
LIN {X 0,Y 711.995,Z 1032.286,A -85,B 0,C 180,E1 32836.022,E2 32836.022} C_VEL
LIN {X 0,Y 712.07,Z 1024.532,A -85,B 0,C 180,E1 32834.359,E2 32834.359} C_VEL
LIN {X 0,Y 712.225,Z 1013.981,A -85,B 0,C 180,E1 32832.411,E2 32832.411} C_VEL
LIN {X 0,Y 712.397,Z 1001.603,A -85,B 0,C 180,E1 32830.486,E2 32830.486} C_VEL
LIN {X 0,Y 712.605,Z 989.787,A -85,B 0,C 180,E1 32828.863,E2 32828.863} C_VEL
LIN {X 0,Y 712.956,Z 974.163,A -85,B 0,C 180,E1 32826.966,E2 32826.966} C_VEL
LIN {X 0,Y 713.304,Z 958.588,A -85,B 0,C 180,E1 32825.309,E2 32825.309} C_VEL
LIN {X 0,Y 713.785,Z 941.053,A -85,B 0,C 180,E1 32823.637,E2 32823.637} C_VEL
LIN {X 0,Y 714.299,Z 921.857,A -85,B 0,C 180,E1 32822.035,E2 32822.035} C_VEL
LIN {X 0,Y 714.883,Z 902.638,A -85,B 0,C 180,E1 32820.598,E2 32820.598} C_VEL
LIN {X 0,Y 715.472,Z 881.199,A -85,B 0,C 180,E1 32819.19,E2 32819.19} C_VEL
LIN {X 0,Y 716.083,Z 861.538,A -85,B 0,C 180,E1 32818.048,E2 32818.048} C_VEL
LIN {X 0,Y 716.784,Z 837.473,A -85,B 0,C 180,E1 32816.823,E2 32816.823} C_VEL
LIN {X 0,Y 717.338,Z 815.668,A -85,B 0,C 180,E1 32815.872,E2 32815.872} C_VEL
LIN {X 0,Y 717.913,Z 793.936,A -85,B 0,C 180,E1 32815.056,E2 32815.056} C_VEL
LIN {X 0,Y 718.524,Z 767.907,A -85,B 0,C 180,E1 32814.244,E2 32814.244} C_VEL
LIN {X 0,Y 718.916,Z 745.225,A -85,B 0,C 180,E1 32813.678,E2 32813.678} C_VEL
LIN {X 0,Y 719.237,Z 723.359,A -85,B 0,C 180,E1 32813.248,E2 32813.248} C_VEL
LIN {X 0,Y 719.58,Z 694.337,A -85,B 0,C 180,E1 32812.844,E2 32812.844} C_VEL
LIN {X 0,Y 720.863,Z 451.6,A -85,B 0,C 180,E1 32810.003,E2 32810.003} C_VEL
LIN {X 0,Y 721.631,Z 289.24,A -85,B 0,C 180,E1 32808.042,E2 32808.042} C_VEL
LIN {X 0,Y 718.682,Z 278.094,A -85,B 0,C 180,E1 32807.705,E2 32807.705} C_VEL
LIN {X 0,Y 718.627,Z 273.586,A -85,B 0,C 180,E1 32807.396,E2 32807.396} C_VEL
LIN {X 0,Y 712.242,Z 257.46,A -85,B 0,C 180,E1 32805.728,E2 32805.728} C_VEL
LIN {X 0,Y 712.204,Z 257.253,A -85,B 0,C 180,E1 32803.228,E2 32803.228} C_VEL
LIN {X 0,Y 712.276,Z 257.251,A -85,B 0,C 180,E1 32800.433,E2 32800.433} C_VEL
LIN {X 0,Y 712.209,Z 257.252,A -85,B 0,C 180,E1 32797.513,E2 32797.513} C_VEL
LIN {X 0,Y 712.207,Z 257.261,A -85,B 0,C 180,E1 32795.044,E2 32795.044} C_VEL
LIN {X 0,Y 712.282,Z 257.256,A -85,B 0,C 180,E1 32792.143,E2 32792.143} C_VEL
LIN {X 0,Y 712.207,Z 257.257,A -85,B 0,C 180,E1 32789.327,E2 32789.327} C_VEL
LIN {X 0,Y 712.207,Z 257.257,A -85,B 0,C 180,E1 32786.876,E2 32786.876} C_VEL
LIN {X 0,Y 712.282,Z 257.257,A -85,B 0,C 180,E1 32783.935,E2 32783.935} C_VEL
LIN {X 0,Y 712.204,Z 257.252,A -85,B 0,C 180,E1 32781.15,E2 32781.15} C_VEL
LIN {X 0,Y 712.215,Z 257.251,A -85,B 0,C 180,E1 32778.624,E2 32778.624} C_VEL
LIN {X 0,Y 712.26,Z 257.25,A -85,B 0,C 180,E1 32775.63,E2 32775.63} C_VEL
LIN {X 0,Y 712.202,Z 257.247,A -85,B 0,C 180,E1 32772.981,E2 32772.981} C_VEL
LIN {X 0,Y 712.22,Z 257.26,A -85,B 0,C 180,E1 32770.434,E2 32770.434} C_VEL
LIN {X 0,Y 712.248,Z 257.238,A -85,B 0,C 180,E1 32767.421,E2 32767.421} C_VEL
LIN {X 0,Y 712.203,Z 257.255,A -85,B 0,C 180,E1 32764.751,E2 32764.751} C_VEL
LIN {X 0,Y 712.242,Z 257.26,A -85,B 0,C 180,E1 32762.092,E2 32762.092} C_VEL
LIN {X 0,Y 712.221,Z 257.249,A -85,B 0,C 180,E1 32759.035,E2 32759.035} C_VEL
LIN {X 0,Y 712.205,Z 257.259,A -85,B 0,C 180,E1 32756.458,E2 32756.458} C_VEL
LIN {X 0,Y 712.281,Z 257.241,A -85,B 0,C 180,E1 32753.633,E2 32753.633} C_VEL
LIN {X 0,Y 712.207,Z 257.255,A -85,B 0,C 180,E1 32750.709,E2 32750.709} C_VEL
LIN {X 0,Y 712.212,Z 257.258,A -85,B 0,C 180,E1 32748.172,E2 32748.172} C_VEL
LIN {X 0,Y 712.274,Z 257.25,A -85,B 0,C 180,E1 32745.197,E2 32745.197} C_VEL
LIN {X 0,Y 712.204,Z 257.257,A -85,B 0,C 180,E1 32742.415,E2 32742.415} C_VEL
LIN {X 0,Y 712.234,Z 257.248,A -85,B 0,C 180,E1 32739.796,E2 32739.796} C_VEL
LIN {X 0,Y 712.224,Z 257.257,A -85,B 0,C 180,E1 32736.678,E2 32736.678} C_VEL
LIN {X 0,Y 712.205,Z 257.257,A -85,B 0,C 180,E1 32734.111,E2 32734.111} C_VEL
LIN {X 0,Y 712.285,Z 257.256,A -85,B 0,C 180,E1 32731.308,E2 32731.308} C_VEL
LIN {X 0,Y 712.211,Z 257.251,A -85,B 0,C 180,E1 32728.421,E2 32728.421} C_VEL
LIN {X 0,Y 712.207,Z 257.252,A -85,B 0,C 180,E1 32725.926,E2 32725.926} C_VEL
LIN {X 0,Y 712.284,Z 257.245,A -85,B 0,C 180,E1 32723.071,E2 32723.071} C_VEL
LIN {X 0,Y 712.209,Z 257.259,A -85,B 0,C 180,E1 32720.194,E2 32720.194} C_VEL
LIN {X 0,Y 712.216,Z 257.261,A -85,B 0,C 180,E1 32717.633,E2 32717.633} C_VEL
LIN {X 0,Y 712.262,Z 257.248,A -85,B 0,C 180,E1 32714.623,E2 32714.623} C_VEL
LIN {X 0,Y 712.215,Z 257.319,A -85,B 0,C 180,E1 32711.987,E2 32711.987} C_VEL
LIN {X 0,Y 712.448,Z 258.445,A -85,B 0,C 180,E1 32711.808,E2 32711.808} C_VEL
LIN {X 0,Y 718.173,Z 272.156,A -85,B 0,C 180,E1 32710.397,E2 32710.397} C_VEL
LIN {X 0,Y 718.992,Z 274.302,A -85,B 0,C 180,E1 32710.186,E2 32710.186} C_VEL
LIN {X 0,Y 718.808,Z 288.002,A -85,B 0,C 180,E1 32709.245,E2 32709.245} C_VEL
LIN {X 0,Y 721.797,Z 300.373,A -85,B 0,C 180,E1 32708.888,E2 32708.888} C_VEL
LIN {X 0,Y 720.391,Z 548.185,A -85,B 0,C 180,E1 32705.929,E2 32705.929} C_VEL
LIN {X 0,Y 719.442,Z 720.366,A -85,B 0,C 180,E1 32703.905,E2 32703.905} C_VEL
LIN {X 0,Y 719.147,Z 745.311,A -85,B 0,C 180,E1 32703.491,E2 32703.491} C_VEL
LIN {X 0,Y 718.6,Z 770.881,A -85,B 0,C 180,E1 32702.9,E2 32702.9} C_VEL
LIN {X 0,Y 718.166,Z 792.504,A -85,B 0,C 180,E1 32702.277,E2 32702.277} C_VEL
LIN {X 0,Y 717.614,Z 817.526,A -85,B 0,C 180,E1 32701.407,E2 32701.407} C_VEL
LIN {X 0,Y 716.952,Z 840.592,A -85,B 0,C 180,E1 32700.444,E2 32700.444} C_VEL
LIN {X 0,Y 716.346,Z 861.803,A -85,B 0,C 180,E1 32699.425,E2 32699.425} C_VEL
LIN {X 0,Y 715.672,Z 885.862,A -85,B 0,C 180,E1 32698.088,E2 32698.088} C_VEL
LIN {X 0,Y 715.059,Z 905.302,A -85,B 0,C 180,E1 32696.856,E2 32696.856} C_VEL
LIN {X 0,Y 714.483,Z 926.328,A -85,B 0,C 180,E1 32695.355,E2 32695.355} C_VEL
LIN {X 0,Y 713.943,Z 944.752,A -85,B 0,C 180,E1 32693.859,E2 32693.859} C_VEL
LIN {X 0,Y 713.478,Z 962.733,A -85,B 0,C 180,E1 32692.234,E2 32692.234} C_VEL
LIN {X 0,Y 713.037,Z 979.619,A -85,B 0,C 180,E1 32690.489,E2 32690.489} C_VEL
LIN {X 0,Y 712.74,Z 994.026,A -85,B 0,C 180,E1 32688.824,E2 32688.824} C_VEL
LIN {X 0,Y 712.436,Z 1009.117,A -85,B 0,C 180,E1 32686.828,E2 32686.828} C_VEL
LIN {X 0,Y 712.247,Z 1020.3,A -85,B 0,C 180,E1 32685.136,E2 32685.136} C_VEL
LIN {X 0,Y 712.134,Z 1031.334,A -85,B 0,C 180,E1 32683.23,E2 32683.23} C_VEL
LIN {X 0,Y 712.022,Z 1040.879,A -85,B 0,C 180,E1 32681.256,E2 32681.256} C_VEL
LIN {X 0,Y 711.948,Z 1047.571,A -85,B 0,C 180,E1 32679.621,E2 32679.621} C_VEL
LIN {X 0,Y 711.933,Z 1053.403,A -85,B 0,C 180,E1 32677.911,E2 32677.911} C_VEL
LIN {X 0,Y 711.908,Z 1058.885,A -85,B 0,C 180,E1 32675.885,E2 32675.885} C_VEL
LIN {X 0,Y 711.914,Z 1062.563,A -85,B 0,C 180,E1 32673.866,E2 32673.866} C_VEL
LIN {X 0,Y 711.905,Z 1064.505,A -85,B 0,C 180,E1 32672.173,E2 32672.173} C_VEL
LIN {X 0,Y 711.892,Z 1065.395,A -85,B 0,C 180,E1 32670.402,E2 32670.402} C_VEL
LIN {X 0,Y 711.899,Z 1064.841,A -85,B 0,C 180,E1 32668.229,E2 32668.229} C_VEL
LIN {X 0,Y 711.903,Z 1063.014,A -85,B 0,C 180,E1 32666.457,E2 32666.457} C_VEL
LIN {X 0,Y 711.912,Z 1060.144,A -85,B 0,C 180,E1 32664.751,E2 32664.751} C_VEL
LIN {X 0,Y 711.936,Z 1055.586,A -85,B 0,C 180,E1 32662.819,E2 32662.819} C_VEL
LIN {X 0,Y 711.962,Z 1048.791,A -85,B 0,C 180,E1 32660.706,E2 32660.706} C_VEL
LIN {X 0,Y 711.998,Z 1042.011,A -85,B 0,C 180,E1 32659.004,E2 32659.004} C_VEL
LIN {X 0,Y 712.076,Z 1034.247,A -85,B 0,C 180,E1 32657.347,E2 32657.347} C_VEL
LIN {X 0,Y 712.224,Z 1023.408,A -85,B 0,C 180,E1 32655.363,E2 32655.363} C_VEL
LIN {X 0,Y 712.396,Z 1011.6,A -85,B 0,C 180,E1 32653.53,E2 32653.53} C_VEL
LIN {X 0,Y 712.615,Z 999.355,A -85,B 0,C 180,E1 32651.851,E2 32651.851} C_VEL
LIN {X 0,Y 712.96,Z 983.2,A -85,B 0,C 180,E1 32649.904,E2 32649.904} C_VEL
LIN {X 0,Y 713.308,Z 968.426,A -85,B 0,C 180,E1 32648.338,E2 32648.338} C_VEL
LIN {X 0,Y 713.793,Z 950.644,A -85,B 0,C 180,E1 32646.645,E2 32646.645} C_VEL
LIN {X 0,Y 714.299,Z 931.869,A -85,B 0,C 180,E1 32645.081,E2 32645.081} C_VEL
LIN {X 0,Y 714.889,Z 912.537,A -85,B 0,C 180,E1 32643.636,E2 32643.636} C_VEL
LIN {X 0,Y 715.494,Z 890.676,A -85,B 0,C 180,E1 32642.204,E2 32642.204} C_VEL
LIN {X 0,Y 716.097,Z 871.109,A -85,B 0,C 180,E1 32641.07,E2 32641.07} C_VEL
LIN {X 0,Y 716.789,Z 847.2,A -85,B 0,C 180,E1 32639.856,E2 32639.856} C_VEL
LIN {X 0,Y 717.347,Z 825.413,A -85,B 0,C 180,E1 32638.907,E2 32638.907} C_VEL
LIN {X 0,Y 717.923,Z 803.695,A -85,B 0,C 180,E1 32638.093,E2 32638.093} C_VEL
LIN {X 0,Y 718.525,Z 777.777,A -85,B 0,C 180,E1 32637.285,E2 32637.285} C_VEL
LIN {X 0,Y 718.917,Z 755.141,A -85,B 0,C 180,E1 32636.721,E2 32636.721} C_VEL
LIN {X 0,Y 719.239,Z 733.181,A -85,B 0,C 180,E1 32636.29,E2 32636.29} C_VEL
LIN {X 0,Y 719.583,Z 703.299,A -85,B 0,C 180,E1 32635.876,E2 32635.876} C_VEL
LIN {X 0,Y 720.866,Z 461.099,A -85,B 0,C 180,E1 32633.042,E2 32633.042} C_VEL
LIN {X 0,Y 721.651,Z 298.994,A -85,B 0,C 180,E1 32631.085,E2 32631.085} C_VEL
LIN {X 0,Y 718.741,Z 287.462,A -85,B 0,C 180,E1 32630.73,E2 32630.73} C_VEL
LIN {X 0,Y 718.894,Z 273.953,A -85,B 0,C 180,E1 32629.782,E2 32629.782} C_VEL
LIN {X 0,Y 713.529,Z 260.761,A -85,B 0,C 180,E1 32628.445,E2 32628.445} C_VEL
LIN {X 0,Y 712.23,Z 257.437,A -85,B 0,C 180,E1 32628.068,E2 32628.068} C_VEL
LIN {X 0,Y 712.261,Z 257.247,A -85,B 0,C 180,E1 32625.377,E2 32625.377} C_VEL
LIN {X 0,Y 712.215,Z 257.253,A -85,B 0,C 180,E1 32622.368,E2 32622.368} C_VEL
LIN {X 0,Y 712.208,Z 257.258,A -85,B 0,C 180,E1 32619.83,E2 32619.83} C_VEL
LIN {X 0,Y 712.283,Z 257.253,A -85,B 0,C 180,E1 32616.99,E2 32616.99} C_VEL
LIN {X 0,Y 712.211,Z 257.247,A -85,B 0,C 180,E1 32614.165,E2 32614.165} C_VEL
LIN {X 0,Y 712.207,Z 257.258,A -85,B 0,C 180,E1 32611.673,E2 32611.673} C_VEL
LIN {X 0,Y 712.283,Z 257.244,A -85,B 0,C 180,E1 32608.783,E2 32608.783} C_VEL
LIN {X 0,Y 712.209,Z 257.26,A -85,B 0,C 180,E1 32605.978,E2 32605.978} C_VEL
LIN {X 0,Y 712.21,Z 257.254,A -85,B 0,C 180,E1 32603.498,E2 32603.498} C_VEL
LIN {X 0,Y 712.285,Z 257.256,A -85,B 0,C 180,E1 32600.631,E2 32600.631} C_VEL
LIN {X 0,Y 712.207,Z 257.258,A -85,B 0,C 180,E1 32597.822,E2 32597.822} C_VEL
LIN {X 0,Y 712.214,Z 257.256,A -85,B 0,C 180,E1 32595.304,E2 32595.304} C_VEL
LIN {X 0,Y 712.266,Z 257.257,A -85,B 0,C 180,E1 32592.321,E2 32592.321} C_VEL
LIN {X 0,Y 712.204,Z 257.257,A -85,B 0,C 180,E1 32589.617,E2 32589.617} C_VEL
LIN {X 0,Y 712.218,Z 257.255,A -85,B 0,C 180,E1 32587.097,E2 32587.097} C_VEL
LIN {X 0,Y 712.255,Z 257.258,A -85,B 0,C 180,E1 32584.106,E2 32584.106} C_VEL
LIN {X 0,Y 712.203,Z 257.258,A -85,B 0,C 180,E1 32581.448,E2 32581.448} C_VEL
LIN {X 0,Y 712.225,Z 257.254,A -85,B 0,C 180,E1 32578.874,E2 32578.874} C_VEL
LIN {X 0,Y 712.225,Z 257.256,A -85,B 0,C 180,E1 32575.733,E2 32575.733} C_VEL
LIN {X 0,Y 712.202,Z 257.258,A -85,B 0,C 180,E1 32573.227,E2 32573.227} C_VEL
LIN {X 0,Y 712.238,Z 257.251,A -85,B 0,C 180,E1 32570.628,E2 32570.628} C_VEL
LIN {X 0,Y 712.224,Z 257.255,A -85,B 0,C 180,E1 32567.596,E2 32567.596} C_VEL
LIN {X 0,Y 712.203,Z 257.258,A -85,B 0,C 180,E1 32565.029,E2 32565.029} C_VEL
LIN {X 0,Y 712.27,Z 257.25,A -85,B 0,C 180,E1 32562.264,E2 32562.264} C_VEL
LIN {X 0,Y 712.203,Z 257.258,A -85,B 0,C 180,E1 32560.965,E2 32560.965} C_VEL
LIN {X 0,Y 711.218,Z 257.386,A -85,B 0,C 180,E1 32560.345,E2 32560.345} C_VEL
LIN {X 0,Y 704.836,Z 258.173,A -85,B 0,C 180,E1 32558.609,E2 32558.609} C_VEL
LIN {X 0,Y 704.336,Z 258.24,A -85,B 0,C 180,E1 32558.158,E2 32558.158} C_VEL
LIN {X 0,Y 704.271,Z 258.238,A -85,B 0,C 180,E1 32555.239,E2 32555.239} C_VEL
LIN {X 0,Y 704.267,Z 258.232,A -85,B 0,C 180,E1 32552.704,E2 32552.704} C_VEL
LIN {X 0,Y 704.347,Z 258.248,A -85,B 0,C 180,E1 32549.829,E2 32549.829} C_VEL
LIN {X 0,Y 704.263,Z 258.229,A -85,B 0,C 180,E1 32546.962,E2 32546.962} C_VEL
LIN {X 0,Y 704.277,Z 258.246,A -85,B 0,C 180,E1 32544.402,E2 32544.402} C_VEL
LIN {X 0,Y 704.305,Z 258.251,A -85,B 0,C 180,E1 32541.336,E2 32541.336} C_VEL
LIN {X 0,Y 704.263,Z 258.246,A -85,B 0,C 180,E1 32538.682,E2 32538.682} C_VEL
LIN {X 0,Y 704.301,Z 258.244,A -85,B 0,C 180,E1 32536.034,E2 32536.034} C_VEL
LIN {X 0,Y 704.278,Z 258.25,A -85,B 0,C 180,E1 32532.959,E2 32532.959} C_VEL
LIN {X 0,Y 704.262,Z 258.24,A -85,B 0,C 180,E1 32530.447,E2 32530.447} C_VEL
LIN {X 0,Y 704.304,Z 258.521,A -85,B 0,C 180,E1 32528.657,E2 32528.657} C_VEL
LIN {X 0,Y 711.691,Z 277.043,A -85,B 0,C 180,E1 32526.724,E2 32526.724} C_VEL
LIN {X 0,Y 712.297,Z 279.72,A -85,B 0,C 180,E1 32526.599,E2 32526.599} C_VEL
LIN {X 0,Y 715.551,Z 292.667,A -85,B 0,C 180,E1 32526.218,E2 32526.218} C_VEL
LIN {X 0,Y 713.889,Z 541.114,A -85,B 0,C 180,E1 32523.228,E2 32523.228} C_VEL
LIN {X 0,Y 712.787,Z 710.6,A -85,B 0,C 180,E1 32521.217,E2 32521.217} C_VEL
LIN {X 0,Y 712.425,Z 735.994,A -85,B 0,C 180,E1 32520.789,E2 32520.789} C_VEL
LIN {X 0,Y 711.812,Z 761.136,A -85,B 0,C 180,E1 32520.203,E2 32520.203} C_VEL
LIN {X 0,Y 711.288,Z 783.031,A -85,B 0,C 180,E1 32519.565,E2 32519.565} C_VEL
LIN {X 0,Y 710.619,Z 808.335,A -85,B 0,C 180,E1 32518.673,E2 32518.673} C_VEL
LIN {X 0,Y 709.9,Z 830.423,A -85,B 0,C 180,E1 32517.743,E2 32517.743} C_VEL
LIN {X 0,Y 709.182,Z 851.403,A -85,B 0,C 180,E1 32516.728,E2 32516.728} C_VEL
LIN {X 0,Y 708.373,Z 875.743,A -85,B 0,C 180,E1 32515.366,E2 32515.366} C_VEL
LIN {X 0,Y 707.686,Z 894.868,A -85,B 0,C 180,E1 32514.144,E2 32514.144} C_VEL
LIN {X 0,Y 706.997,Z 915.467,A -85,B 0,C 180,E1 32512.668,E2 32512.668} C_VEL
LIN {X 0,Y 706.371,Z 933.917,A -85,B 0,C 180,E1 32511.159,E2 32511.159} C_VEL
LIN {X 0,Y 705.808,Z 950.895,A -85,B 0,C 180,E1 32509.618,E2 32509.618} C_VEL
LIN {X 0,Y 705.319,Z 968.254,A -85,B 0,C 180,E1 32507.831,E2 32507.831} C_VEL
LIN {X 0,Y 704.925,Z 982.338,A -85,B 0,C 180,E1 32506.202,E2 32506.202} C_VEL
LIN {X 0,Y 704.588,Z 997.298,A -85,B 0,C 180,E1 32504.243,E2 32504.243} C_VEL
LIN {X 0,Y 704.355,Z 1009.479,A -85,B 0,C 180,E1 32502.398,E2 32502.398} C_VEL
LIN {X 0,Y 704.181,Z 1019.69,A -85,B 0,C 180,E1 32500.637,E2 32500.637} C_VEL
LIN {X 0,Y 704.061,Z 1030.222,A -85,B 0,C 180,E1 32498.493,E2 32498.493} C_VEL
LIN {X 0,Y 703.964,Z 1037.26,A -85,B 0,C 180,E1 32496.77,E2 32496.77} C_VEL
LIN {X 0,Y 703.944,Z 1043.106,A -85,B 0,C 180,E1 32495.052,E2 32495.052} C_VEL
LIN {X 0,Y 703.922,Z 1048.214,A -85,B 0,C 180,E1 32493.176,E2 32493.176} C_VEL
LIN {X 0,Y 703.917,Z 1052.408,A -85,B 0,C 180,E1 32490.977,E2 32490.977} C_VEL
LIN {X 0,Y 703.9,Z 1054.411,A -85,B 0,C 180,E1 32489.267,E2 32489.267} C_VEL
LIN {X 0,Y 703.892,Z 1055.341,A -85,B 0,C 180,E1 32487.558,E2 32487.558} C_VEL
LIN {X 0,Y 703.906,Z 1055.134,A -85,B 0,C 180,E1 32485.601,E2 32485.601} C_VEL
LIN {X 0,Y 703.904,Z 1053.271,A -85,B 0,C 180,E1 32483.557,E2 32483.557} C_VEL
LIN {X 0,Y 703.915,Z 1050.35,A -85,B 0,C 180,E1 32481.751,E2 32481.751} C_VEL
LIN {X 0,Y 703.926,Z 1046.414,A -85,B 0,C 180,E1 32480.021,E2 32480.021} C_VEL
LIN {X 0,Y 703.964,Z 1040.242,A -85,B 0,C 180,E1 32477.948,E2 32477.948} C_VEL
LIN {X 0,Y 704.011,Z 1032.851,A -85,B 0,C 180,E1 32476.028,E2 32476.028} C_VEL
LIN {X 0,Y 704.099,Z 1025.101,A -85,B 0,C 180,E1 32474.33,E2 32474.33} C_VEL
LIN {X 0,Y 704.253,Z 1015.781,A -85,B 0,C 180,E1 32472.568,E2 32472.568} C_VEL
LIN {X 0,Y 704.481,Z 1002.527,A -85,B 0,C 180,E1 32470.43,E2 32470.43} C_VEL
LIN {X 0,Y 704.738,Z 990.156,A -85,B 0,C 180,E1 32468.702,E2 32468.702} C_VEL
LIN {X 0,Y 705.133,Z 975.387,A -85,B 0,C 180,E1 32466.872,E2 32466.872} C_VEL
LIN {X 0,Y 705.573,Z 959.075,A -85,B 0,C 180,E1 32465.109,E2 32465.109} C_VEL
LIN {X 0,Y 706.101,Z 942.061,A -85,B 0,C 180,E1 32463.463,E2 32463.463} C_VEL
LIN {X 0,Y 706.732,Z 922.674,A -85,B 0,C 180,E1 32461.815,E2 32461.815} C_VEL
LIN {X 0,Y 707.365,Z 904.58,A -85,B 0,C 180,E1 32460.441,E2 32460.441} C_VEL
LIN {X 0,Y 708.128,Z 882.039,A -85,B 0,C 180,E1 32458.93,E2 32458.93} C_VEL
LIN {X 0,Y 708.827,Z 862.467,A -85,B 0,C 180,E1 32457.777,E2 32457.777} C_VEL
LIN {X 0,Y 709.641,Z 839.217,A -85,B 0,C 180,E1 32456.57,E2 32456.57} C_VEL
LIN {X 0,Y 710.339,Z 815.821,A -85,B 0,C 180,E1 32455.538,E2 32455.538} C_VEL
LIN {X 0,Y 710.984,Z 794.772,A -85,B 0,C 180,E1 32454.739,E2 32454.739} C_VEL
LIN {X 0,Y 711.701,Z 768.871,A -85,B 0,C 180,E1 32453.917,E2 32453.917} C_VEL
LIN {X 0,Y 712.172,Z 745.369,A -85,B 0,C 180,E1 32453.325,E2 32453.325} C_VEL
LIN {X 0,Y 712.556,Z 723.244,A -85,B 0,C 180,E1 32452.887,E2 32452.887} C_VEL
LIN {X 0,Y 712.956,Z 693.378,A -85,B 0,C 180,E1 32452.471,E2 32452.471} C_VEL
LIN {X 0,Y 714.462,Z 451.56,A -85,B 0,C 180,E1 32449.615,E2 32449.615} C_VEL
LIN {X 0,Y 715.394,Z 291.261,A -85,B 0,C 180,E1 32447.663,E2 32447.663} C_VEL
LIN {X 0,Y 711.877,Z 277.809,A -85,B 0,C 180,E1 32447.244,E2 32447.244} C_VEL
LIN {X 0,Y 706.456,Z 264.093,A -85,B 0,C 180,E1 32445.856,E2 32445.856} C_VEL
LIN {X 0,Y 704.29,Z 258.42,A -85,B 0,C 180,E1 32445.231,E2 32445.231} C_VEL
LIN {X 0,Y 704.335,Z 258.241,A -85,B 0,C 180,E1 32442.512,E2 32442.512} C_VEL
LIN {X 0,Y 704.271,Z 258.25,A -85,B 0,C 180,E1 32439.563,E2 32439.563} C_VEL
LIN {X 0,Y 704.267,Z 258.242,A -85,B 0,C 180,E1 32437.07,E2 32437.07} C_VEL
LIN {X 0,Y 704.345,Z 258.238,A -85,B 0,C 180,E1 32434.206,E2 32434.206} C_VEL
LIN {X 0,Y 704.27,Z 258.245,A -85,B 0,C 180,E1 32431.403,E2 32431.403} C_VEL
LIN {X 0,Y 704.271,Z 258.248,A -85,B 0,C 180,E1 32428.863,E2 32428.863} C_VEL
LIN {X 0,Y 704.335,Z 258.23,A -85,B 0,C 180,E1 32425.928,E2 32425.928} C_VEL
LIN {X 0,Y 704.266,Z 258.248,A -85,B 0,C 180,E1 32423.159,E2 32423.159} C_VEL
LIN {X 0,Y 704.279,Z 258.243,A -85,B 0,C 180,E1 32420.616,E2 32420.616} C_VEL
LIN {X 0,Y 704.312,Z 258.245,A -85,B 0,C 180,E1 32417.601,E2 32417.601} C_VEL
LIN {X 0,Y 704.263,Z 258.241,A -85,B 0,C 180,E1 32414.975,E2 32414.975} C_VEL
LIN {X 0,Y 704.288,Z 258.237,A -85,B 0,C 180,E1 32412.377,E2 32412.377} C_VEL
LIN {X 0,Y 704.284,Z 258.242,A -85,B 0,C 180,E1 32409.232,E2 32409.232} C_VEL
LIN {X 0,Y 704.263,Z 258.227,A -85,B 0,C 180,E1 32406.686,E2 32406.686} C_VEL
LIN {X 0,Y 704.332,Z 258.248,A -85,B 0,C 180,E1 32403.907,E2 32403.907} C_VEL
LIN {X 0,Y 704.274,Z 258.233,A -85,B 0,C 180,E1 32400.976,E2 32400.976} C_VEL
LIN {X 0,Y 704.267,Z 258.239,A -85,B 0,C 180,E1 32398.454,E2 32398.454} C_VEL
LIN {X 0,Y 704.345,Z 258.242,A -85,B 0,C 180,E1 32395.603,E2 32395.603} C_VEL
LIN {X 0,Y 704.267,Z 258.228,A -85,B 0,C 180,E1 32392.741,E2 32392.741} C_VEL
LIN {X 0,Y 704.274,Z 258.246,A -85,B 0,C 180,E1 32390.191,E2 32390.191} C_VEL
LIN {X 0,Y 704.327,Z 258.228,A -85,B 0,C 180,E1 32387.205,E2 32387.205} C_VEL
LIN {X 0,Y 704.265,Z 258.241,A -85,B 0,C 180,E1 32384.435,E2 32384.435} C_VEL
LIN {X 0,Y 704.303,Z 258.249,A -85,B 0,C 180,E1 32381.762,E2 32381.762} C_VEL
LIN {X 0,Y 704.282,Z 258.239,A -85,B 0,C 180,E1 32378.688,E2 32378.688} C_VEL
LIN {X 0,Y 704.268,Z 258.249,A -85,B 0,C 180,E1 32376.109,E2 32376.109} C_VEL
LIN {X 0,Y 704.347,Z 258.247,A -85,B 0,C 180,E1 32373.243,E2 32373.243} C_VEL
LIN {X 0,Y 704.272,Z 258.248,A -85,B 0,C 180,E1 32370.391,E2 32370.391} C_VEL
LIN {X 0,Y 704.273,Z 258.241,A -85,B 0,C 180,E1 32367.832,E2 32367.832} C_VEL
LIN {X 0,Y 704.33,Z 258.246,A -85,B 0,C 180,E1 32364.856,E2 32364.856} C_VEL
LIN {X 0,Y 704.265,Z 258.232,A -85,B 0,C 180,E1 32362.128,E2 32362.128} C_VEL
LIN {X 0,Y 704.288,Z 258.251,A -85,B 0,C 180,E1 32359.548,E2 32359.548} C_VEL
LIN {X 0,Y 704.288,Z 258.247,A -85,B 0,C 180,E1 32356.371,E2 32356.371} C_VEL
LIN {X 0,Y 704.264,Z 258.24,A -85,B 0,C 180,E1 32353.843,E2 32353.843} C_VEL
LIN {X 0,Y 704.334,Z 258.492,A -85,B 0,C 180,E1 32352.421,E2 32352.421} C_VEL
LIN {X 0,Y 711.997,Z 277.439,A -85,B 0,C 180,E1 32350.433,E2 32350.433} C_VEL
LIN {X 0,Y 712.066,Z 288.033,A -85,B 0,C 180,E1 32349.69,E2 32349.69} C_VEL
LIN {X 0,Y 715.55,Z 302.356,A -85,B 0,C 180,E1 32349.267,E2 32349.267} C_VEL
LIN {X 0,Y 713.898,Z 549.712,A -85,B 0,C 180,E1 32346.289,E2 32346.289} C_VEL
LIN {X 0,Y 712.788,Z 720.498,A -85,B 0,C 180,E1 32344.264,E2 32344.264} C_VEL
LIN {X 0,Y 712.433,Z 745.754,A -85,B 0,C 180,E1 32343.839,E2 32343.839} C_VEL
LIN {X 0,Y 711.812,Z 771.107,A -85,B 0,C 180,E1 32343.248,E2 32343.248} C_VEL
LIN {X 0,Y 711.297,Z 792.508,A -85,B 0,C 180,E1 32342.627,E2 32342.627} C_VEL
LIN {X 0,Y 710.65,Z 817.523,A -85,B 0,C 180,E1 32341.75,E2 32341.75} C_VEL
LIN {X 0,Y 709.906,Z 840.246,A -85,B 0,C 180,E1 32340.796,E2 32340.796} C_VEL
LIN {X 0,Y 709.199,Z 860.869,A -85,B 0,C 180,E1 32339.801,E2 32339.801} C_VEL
LIN {X 0,Y 708.422,Z 884.39,A -85,B 0,C 180,E1 32338.494,E2 32338.494} C_VEL
LIN {X 0,Y 707.718,Z 904.074,A -85,B 0,C 180,E1 32337.242,E2 32337.242} C_VEL
LIN {X 0,Y 707.023,Z 924.617,A -85,B 0,C 180,E1 32335.779,E2 32335.779} C_VEL
LIN {X 0,Y 706.365,Z 944.055,A -85,B 0,C 180,E1 32334.192,E2 32334.192} C_VEL
LIN {X 0,Y 705.799,Z 961.253,A -85,B 0,C 180,E1 32332.629,E2 32332.629} C_VEL
LIN {X 0,Y 705.31,Z 978.539,A -85,B 0,C 180,E1 32330.844,E2 32330.844} C_VEL
LIN {X 0,Y 704.92,Z 992.618,A -85,B 0,C 180,E1 32329.213,E2 32329.213} C_VEL
LIN {X 0,Y 704.578,Z 1007.64,A -85,B 0,C 180,E1 32327.238,E2 32327.238} C_VEL
LIN {X 0,Y 704.355,Z 1019.488,A -85,B 0,C 180,E1 32325.442,E2 32325.442} C_VEL
LIN {X 0,Y 704.183,Z 1029.495,A -85,B 0,C 180,E1 32323.717,E2 32323.717} C_VEL
LIN {X 0,Y 704.061,Z 1040.168,A -85,B 0,C 180,E1 32321.551,E2 32321.551} C_VEL
LIN {X 0,Y 703.963,Z 1047.267,A -85,B 0,C 180,E1 32319.814,E2 32319.814} C_VEL
LIN {X 0,Y 703.943,Z 1053.148,A -85,B 0,C 180,E1 32318.084,E2 32318.084} C_VEL
LIN {X 0,Y 703.924,Z 1058.273,A -85,B 0,C 180,E1 32316.197,E2 32316.197} C_VEL
LIN {X 0,Y 703.913,Z 1062.45,A -85,B 0,C 180,E1 32313.991,E2 32313.991} C_VEL
LIN {X 0,Y 703.905,Z 1064.506,A -85,B 0,C 180,E1 32312.198,E2 32312.198} C_VEL
LIN {X 0,Y 703.892,Z 1065.395,A -85,B 0,C 180,E1 32310.407,E2 32310.407} C_VEL
LIN {X 0,Y 703.9,Z 1064.841,A -85,B 0,C 180,E1 32308.209,E2 32308.209} C_VEL
LIN {X 0,Y 703.905,Z 1063.014,A -85,B 0,C 180,E1 32306.417,E2 32306.417} C_VEL
LIN {X 0,Y 703.91,Z 1060.166,A -85,B 0,C 180,E1 32304.702,E2 32304.702} C_VEL
LIN {X 0,Y 703.938,Z 1055.793,A -85,B 0,C 180,E1 32302.819,E2 32302.819} C_VEL
LIN {X 0,Y 703.97,Z 1049.096,A -85,B 0,C 180,E1 32300.682,E2 32300.682} C_VEL
LIN {X 0,Y 704.019,Z 1042.251,A -85,B 0,C 180,E1 32298.934,E2 32298.934} C_VEL
LIN {X 0,Y 704.118,Z 1034.248,A -85,B 0,C 180,E1 32297.201,E2 32297.201} C_VEL
LIN {X 0,Y 704.279,Z 1023.407,A -85,B 0,C 180,E1 32295.194,E2 32295.194} C_VEL
LIN {X 0,Y 704.498,Z 1011.602,A -85,B 0,C 180,E1 32293.34,E2 32293.34} C_VEL
LIN {X 0,Y 704.761,Z 999.357,A -85,B 0,C 180,E1 32291.641,E2 32291.641} C_VEL
LIN {X 0,Y 705.162,Z 983.198,A -85,B 0,C 180,E1 32289.672,E2 32289.672} C_VEL
LIN {X 0,Y 705.585,Z 968.717,A -85,B 0,C 180,E1 32288.118,E2 32288.118} C_VEL
LIN {X 0,Y 706.133,Z 951.126,A -85,B 0,C 180,E1 32286.421,E2 32286.421} C_VEL
LIN {X 0,Y 706.74,Z 932.423,A -85,B 0,C 180,E1 32284.84,E2 32284.84} C_VEL
LIN {X 0,Y 707.375,Z 914.359,A -85,B 0,C 180,E1 32283.47,E2 32283.47} C_VEL
LIN {X 0,Y 708.149,Z 891.538,A -85,B 0,C 180,E1 32281.944,E2 32281.944} C_VEL
LIN {X 0,Y 708.851,Z 871.835,A -85,B 0,C 180,E1 32280.787,E2 32280.787} C_VEL
LIN {X 0,Y 709.657,Z 848.371,A -85,B 0,C 180,E1 32279.576,E2 32279.576} C_VEL
LIN {X 0,Y 710.358,Z 825.416,A -85,B 0,C 180,E1 32278.567,E2 32278.567} C_VEL
LIN {X 0,Y 710.978,Z 804.977,A -85,B 0,C 180,E1 32277.791,E2 32277.791} C_VEL
LIN {X 0,Y 711.697,Z 779.177,A -85,B 0,C 180,E1 32276.971,E2 32276.971} C_VEL
LIN {X 0,Y 712.17,Z 755.522,A -85,B 0,C 180,E1 32276.373,E2 32276.373} C_VEL
LIN {X 0,Y 712.552,Z 733.504,A -85,B 0,C 180,E1 32275.936,E2 32275.936} C_VEL
LIN {X 0,Y 712.947,Z 704.698,A -85,B 0,C 180,E1 32275.531,E2 32275.531} C_VEL
LIN {X 0,Y 714.461,Z 462.118,A -85,B 0,C 180,E1 32272.667,E2 32272.667} C_VEL
LIN {X 0,Y 715.429,Z 301.061,A -85,B 0,C 180,E1 32270.708,E2 32270.708} C_VEL
LIN {X 0,Y 711.995,Z 287.479,A -85,B 0,C 180,E1 32270.285,E2 32270.285} C_VEL
LIN {X 0,Y 711.998,Z 277.437,A -85,B 0,C 180,E1 32269.566,E2 32269.566} C_VEL
LIN {X 0,Y 705.606,Z 261.778,A -85,B 0,C 180,E1 32267.949,E2 32267.949} C_VEL
LIN {X 0,Y 704.322,Z 258.373,A -85,B 0,C 180,E1 32267.548,E2 32267.548} C_VEL
LIN {X 0,Y 704.289,Z 258.254,A -85,B 0,C 180,E1 32264.535,E2 32264.535} C_VEL
LIN {X 0,Y 704.267,Z 258.243,A -85,B 0,C 180,E1 32261.931,E2 32261.931} C_VEL
LIN {X 0,Y 704.343,Z 258.233,A -85,B 0,C 180,E1 32259.073,E2 32259.073} C_VEL
LIN {X 0,Y 704.274,Z 258.249,A -85,B 0,C 180,E1 32256.201,E2 32256.201} C_VEL
LIN {X 0,Y 704.273,Z 258.232,A -85,B 0,C 180,E1 32253.622,E2 32253.622} C_VEL
LIN {X 0,Y 704.334,Z 258.245,A -85,B 0,C 180,E1 32250.64,E2 32250.64} C_VEL
LIN {X 0,Y 704.267,Z 258.24,A -85,B 0,C 180,E1 32247.939,E2 32247.939} C_VEL
LIN {X 0,Y 704.281,Z 258.247,A -85,B 0,C 180,E1 32245.389,E2 32245.389} C_VEL
LIN {X 0,Y 704.311,Z 258.25,A -85,B 0,C 180,E1 32242.363,E2 32242.363} C_VEL
LIN {X 0,Y 704.264,Z 258.246,A -85,B 0,C 180,E1 32239.729,E2 32239.729} C_VEL
LIN {X 0,Y 704.298,Z 258.244,A -85,B 0,C 180,E1 32237.09,E2 32237.09} C_VEL
LIN {X 0,Y 704.289,Z 258.248,A -85,B 0,C 180,E1 32234.05,E2 32234.05} C_VEL
LIN {X 0,Y 704.266,Z 258.246,A -85,B 0,C 180,E1 32231.465,E2 32231.465} C_VEL
LIN {X 0,Y 704.337,Z 258.243,A -85,B 0,C 180,E1 32228.655,E2 32228.655} C_VEL
LIN {X 0,Y 704.276,Z 258.248,A -85,B 0,C 180,E1 32225.785,E2 32225.785} C_VEL
LIN {X 0,Y 704.266,Z 258.245,A -85,B 0,C 180,E1 32223.256,E2 32223.256} C_VEL
LIN {X 0,Y 704.347,Z 258.244,A -85,B 0,C 180,E1 32220.407,E2 32220.407} C_VEL
LIN {X 0,Y 704.27,Z 258.248,A -85,B 0,C 180,E1 32217.559,E2 32217.559} C_VEL
LIN {X 0,Y 704.269,Z 258.242,A -85,B 0,C 180,E1 32215.032,E2 32215.032} C_VEL
LIN {X 0,Y 704.342,Z 258.244,A -85,B 0,C 180,E1 32212.085,E2 32212.085} C_VEL
LIN {X 0,Y 704.264,Z 258.248,A -85,B 0,C 180,E1 32209.256,E2 32209.256} C_VEL
LIN {X 0,Y 704.283,Z 258.24,A -85,B 0,C 180,E1 32206.703,E2 32206.703} C_VEL
LIN {X 0,Y 704.291,Z 258.243,A -85,B 0,C 180,E1 32203.589,E2 32203.589} C_VEL
LIN {X 0,Y 704.264,Z 258.248,A -85,B 0,C 180,E1 32200.964,E2 32200.964} C_VEL
LIN {X 0,Y 704.336,Z 258.24,A -85,B 0,C 180,E1 32198.158,E2 32198.158} C_VEL
LIN {X 0,Y 703.384,Z 258.367,A -85,B 0,C 180,E1 32197.531,E2 32197.531} C_VEL
LIN {X 0,Y 696.91,Z 259.166,A -85,B 0,C 180,E1 32195.777,E2 32195.777} C_VEL
LIN {X 0,Y 696.339,Z 259.226,A -85,B 0,C 180,E1 32195.32,E2 32195.32} C_VEL
LIN {X 0,Y 696.327,Z 259.22,A -85,B 0,C 180,E1 32192.729,E2 32192.729} C_VEL
LIN {X 0,Y 696.408,Z 259.237,A -85,B 0,C 180,E1 32189.807,E2 32189.807} C_VEL
LIN {X 0,Y 696.323,Z 259.215,A -85,B 0,C 180,E1 32186.93,E2 32186.93} C_VEL
LIN {X 0,Y 696.344,Z 259.235,A -85,B 0,C 180,E1 32184.339,E2 32184.339} C_VEL
LIN {X 0,Y 696.354,Z 259.241,A -85,B 0,C 180,E1 32181.232,E2 32181.232} C_VEL
LIN {X 0,Y 696.324,Z 259.234,A -85,B 0,C 180,E1 32178.659,E2 32178.659} C_VEL
LIN {X 0,Y 696.37,Z 259.231,A -85,B 0,C 180,E1 32175.976,E2 32175.976} C_VEL
LIN {X 0,Y 696.337,Z 259.238,A -85,B 0,C 180,E1 32172.918,E2 32172.918} C_VEL
LIN {X 0,Y 696.326,Z 259.228,A -85,B 0,C 180,E1 32170.362,E2 32170.362} C_VEL
LIN {X 0,Y 696.406,Z 259.497,A -85,B 0,C 180,E1 32169.165,E2 32169.165} C_VEL
LIN {X 0,Y 703.751,Z 277.831,A -85,B 0,C 180,E1 32167.214,E2 32167.214} C_VEL
LIN {X 0,Y 706.373,Z 282.737,A -85,B 0,C 180,E1 32166.959,E2 32166.959} C_VEL
LIN {X 0,Y 709.334,Z 294.658,A -85,B 0,C 180,E1 32166.604,E2 32166.604} C_VEL
LIN {X 0,Y 707.424,Z 542.499,A -85,B 0,C 180,E1 32163.596,E2 32163.596} C_VEL
LIN {X 0,Y 706.163,Z 710.633,A -85,B 0,C 180,E1 32161.584,E2 32161.584} C_VEL
LIN {X 0,Y 705.74,Z 736.246,A -85,B 0,C 180,E1 32161.148,E2 32161.148} C_VEL
LIN {X 0,Y 705.072,Z 760.959,A -85,B 0,C 180,E1 32160.567,E2 32160.567} C_VEL
LIN {X 0,Y 704.451,Z 782.842,A -85,B 0,C 180,E1 32159.928,E2 32159.928} C_VEL
LIN {X 0,Y 703.682,Z 808.187,A -85,B 0,C 180,E1 32159.029,E2 32159.029} C_VEL
LIN {X 0,Y 702.871,Z 830.298,A -85,B 0,C 180,E1 32158.091,E2 32158.091} C_VEL
LIN {X 0,Y 702.051,Z 851.298,A -85,B 0,C 180,E1 32157.068,E2 32157.068} C_VEL
LIN {X 0,Y 701.096,Z 875.655,A -85,B 0,C 180,E1 32155.693,E2 32155.693} C_VEL
LIN {X 0,Y 700.321,Z 894.793,A -85,B 0,C 180,E1 32154.459,E2 32154.459} C_VEL
LIN {X 0,Y 699.499,Z 915.404,A -85,B 0,C 180,E1 32152.969,E2 32152.969} C_VEL
LIN {X 0,Y 698.766,Z 934.357,A -85,B 0,C 180,E1 32151.401,E2 32151.401} C_VEL
LIN {X 0,Y 698.128,Z 951.295,A -85,B 0,C 180,E1 32149.843,E2 32149.843} C_VEL
LIN {X 0,Y 697.553,Z 968.594,A -85,B 0,C 180,E1 32148.036,E2 32148.036} C_VEL
LIN {X 0,Y 697.083,Z 983.137,A -85,B 0,C 180,E1 32146.328,E2 32146.328} C_VEL
LIN {X 0,Y 696.677,Z 998.338,A -85,B 0,C 180,E1 32144.292,E2 32144.292} C_VEL
LIN {X 0,Y 696.425,Z 1009.99,A -85,B 0,C 180,E1 32142.495,E2 32142.495} C_VEL
LIN {X 0,Y 696.218,Z 1021.246,A -85,B 0,C 180,E1 32140.509,E2 32140.509} C_VEL
LIN {X 0,Y 696.072,Z 1031.081,A -85,B 0,C 180,E1 32138.425,E2 32138.425} C_VEL
LIN {X 0,Y 695.97,Z 1037.996,A -85,B 0,C 180,E1 32136.683,E2 32136.683} C_VEL
LIN {X 0,Y 695.945,Z 1043.975,A -85,B 0,C 180,E1 32134.863,E2 32134.863} C_VEL
LIN {X 0,Y 695.901,Z 1049.547,A -85,B 0,C 180,E1 32132.635,E2 32132.635} C_VEL
LIN {X 0,Y 695.918,Z 1052.681,A -85,B 0,C 180,E1 32130.823,E2 32130.823} C_VEL
LIN {X 0,Y 695.909,Z 1054.574,A -85,B 0,C 180,E1 32129.094,E2 32129.094} C_VEL
LIN {X 0,Y 695.908,Z 1055.484,A -85,B 0,C 180,E1 32127.035,E2 32127.035} C_VEL
LIN {X 0,Y 695.911,Z 1054.634,A -85,B 0,C 180,E1 32124.889,E2 32124.889} C_VEL
LIN {X 0,Y 695.915,Z 1052.75,A -85,B 0,C 180,E1 32123.137,E2 32123.137} C_VEL
LIN {X 0,Y 695.902,Z 1049.479,A -85,B 0,C 180,E1 32121.24,E2 32121.24} C_VEL
LIN {X 0,Y 695.944,Z 1044.038,A -85,B 0,C 180,E1 32119.068,E2 32119.068} C_VEL
LIN {X 0,Y 695.968,Z 1038.246,A -85,B 0,C 180,E1 32117.296,E2 32117.296} C_VEL
LIN {X 0,Y 696.063,Z 1031.616,A -85,B 0,C 180,E1 32115.611,E2 32115.611} C_VEL
LIN {X 0,Y 696.204,Z 1022.517,A -85,B 0,C 180,E1 32113.651,E2 32113.651} C_VEL
LIN {X 0,Y 696.398,Z 1011.039,A -85,B 0,C 180,E1 32111.586,E2 32111.586} C_VEL
LIN {X 0,Y 696.639,Z 999.795,A -85,B 0,C 180,E1 32109.834,E2 32109.834} C_VEL
LIN {X 0,Y 697.025,Z 985.903,A -85,B 0,C 180,E1 32107.924,E2 32107.924} C_VEL
LIN {X 0,Y 697.457,Z 971.1,A -85,B 0,C 180,E1 32106.154,E2 32106.154} C_VEL
LIN {X 0,Y 697.983,Z 955.523,A -85,B 0,C 180,E1 32104.489,E2 32104.489} C_VEL
LIN {X 0,Y 698.68,Z 936.692,A -85,B 0,C 180,E1 32102.714,E2 32102.714} C_VEL
LIN {X 0,Y 699.326,Z 919.72,A -85,B 0,C 180,E1 32101.288,E2 32101.288} C_VEL
LIN {X 0,Y 700.15,Z 898.87,A -85,B 0,C 180,E1 32099.727,E2 32099.727} C_VEL
LIN {X 0,Y 700.96,Z 879.144,A -85,B 0,C 180,E1 32098.432,E2 32098.432} C_VEL
LIN {X 0,Y 701.761,Z 859.233,A -85,B 0,C 180,E1 32097.267,E2 32097.267} C_VEL
LIN {X 0,Y 702.706,Z 834.232,A -85,B 0,C 180,E1 32095.999,E2 32095.999} C_VEL
LIN {X 0,Y 703.473,Z 813.538,A -85,B 0,C 180,E1 32095.098,E2 32095.098} C_VEL
LIN {X 0,Y 704.263,Z 790.98,A -85,B 0,C 180,E1 32094.251,E2 32094.251} C_VEL
LIN {X 0,Y 704.968,Z 764.953,A -85,B 0,C 180,E1 32093.45,E2 32093.45} C_VEL
LIN {X 0,Y 705.506,Z 743.016,A -85,B 0,C 180,E1 32092.909,E2 32092.909} C_VEL
LIN {X 0,Y 706.099,Z 717.447,A -85,B 0,C 180,E1 32092.422,E2 32092.422} C_VEL
LIN {X 0,Y 706.465,Z 677.311,A -85,B 0,C 180,E1 32091.913,E2 32091.913} C_VEL
LIN {X 0,Y 708.134,Z 444.631,A -85,B 0,C 180,E1 32089.136,E2 32089.136} C_VEL
LIN {X 0,Y 709.19,Z 293.316,A -85,B 0,C 180,E1 32087.279,E2 32087.279} C_VEL
LIN {X 0,Y 705.817,Z 281.339,A -85,B 0,C 180,E1 32086.895,E2 32086.895} C_VEL
LIN {X 0,Y 703.577,Z 277.38,A -85,B 0,C 180,E1 32086.653,E2 32086.653} C_VEL
LIN {X 0,Y 697.491,Z 262.511,A -85,B 0,C 180,E1 32085.087,E2 32085.087} C_VEL
LIN {X 0,Y 696.391,Z 259.351,A -85,B 0,C 180,E1 32084.706,E2 32084.706} C_VEL
LIN {X 0,Y 696.337,Z 259.241,A -85,B 0,C 180,E1 32081.67,E2 32081.67} C_VEL
LIN {X 0,Y 696.328,Z 259.241,A -85,B 0,C 180,E1 32079.158,E2 32079.158} C_VEL
LIN {X 0,Y 696.406,Z 259.236,A -85,B 0,C 180,E1 32076.267,E2 32076.267} C_VEL
LIN {X 0,Y 696.329,Z 259.234,A -85,B 0,C 180,E1 32073.365,E2 32073.365} C_VEL
LIN {X 0,Y 696.336,Z 259.236,A -85,B 0,C 180,E1 32070.831,E2 32070.831} C_VEL
LIN {X 0,Y 696.379,Z 259.231,A -85,B 0,C 180,E1 32067.813,E2 32067.813} C_VEL
LIN {X 0,Y 696.323,Z 259.224,A -85,B 0,C 180,E1 32065.063,E2 32065.063} C_VEL
LIN {X 0,Y 696.372,Z 259.24,A -85,B 0,C 180,E1 32062.365,E2 32062.365} C_VEL
LIN {X 0,Y 696.342,Z 259.224,A -85,B 0,C 180,E1 32059.371,E2 32059.371} C_VEL
LIN {X 0,Y 696.329,Z 259.238,A -85,B 0,C 180,E1 32056.776,E2 32056.776} C_VEL
LIN {X 0,Y 696.406,Z 259.214,A -85,B 0,C 180,E1 32053.873,E2 32053.873} C_VEL
LIN {X 0,Y 696.329,Z 259.235,A -85,B 0,C 180,E1 32051.01,E2 32051.01} C_VEL
LIN {X 0,Y 696.341,Z 259.234,A -85,B 0,C 180,E1 32048.422,E2 32048.422} C_VEL
LIN {X 0,Y 696.367,Z 259.23,A -85,B 0,C 180,E1 32045.355,E2 32045.355} C_VEL
LIN {X 0,Y 696.326,Z 259.236,A -85,B 0,C 180,E1 32042.716,E2 32042.716} C_VEL
LIN {X 0,Y 696.37,Z 259.217,A -85,B 0,C 180,E1 32040,E2 32040} C_VEL
LIN {X 0,Y 696.34,Z 259.235,A -85,B 0,C 180,E1 32036.954,E2 32036.954} C_VEL
LIN {X 0,Y 696.328,Z 259.231,A -85,B 0,C 180,E1 32034.396,E2 32034.396} C_VEL
LIN {X 0,Y 696.406,Z 259.224,A -85,B 0,C 180,E1 32031.496,E2 32031.496} C_VEL
LIN {X 0,Y 696.331,Z 259.233,A -85,B 0,C 180,E1 32028.654,E2 32028.654} C_VEL
LIN {X 0,Y 696.337,Z 259.218,A -85,B 0,C 180,E1 32026.092,E2 32026.092} C_VEL
LIN {X 0,Y 696.377,Z 259.233,A -85,B 0,C 180,E1 32023.054,E2 32023.054} C_VEL
LIN {X 0,Y 696.326,Z 259.223,A -85,B 0,C 180,E1 32020.366,E2 32020.366} C_VEL
LIN {X 0,Y 696.36,Z 259.232,A -85,B 0,C 180,E1 32017.724,E2 32017.724} C_VEL
LIN {X 0,Y 696.347,Z 259.233,A -85,B 0,C 180,E1 32014.665,E2 32014.665} C_VEL
LIN {X 0,Y 696.329,Z 259.236,A -85,B 0,C 180,E1 32012.088,E2 32012.088} C_VEL
LIN {X 0,Y 696.401,Z 259.231,A -85,B 0,C 180,E1 32009.26,E2 32009.26} C_VEL
LIN {X 0,Y 696.332,Z 259.226,A -85,B 0,C 180,E1 32006.339,E2 32006.339} C_VEL
LIN {X 0,Y 696.339,Z 259.24,A -85,B 0,C 180,E1 32003.729,E2 32003.729} C_VEL
LIN {X 0,Y 696.381,Z 259.228,A -85,B 0,C 180,E1 32000.707,E2 32000.707} C_VEL
LIN {X 0,Y 696.328,Z 259.238,A -85,B 0,C 180,E1 31997.998,E2 31997.998} C_VEL
LIN {X 0,Y 696.37,Z 259.242,A -85,B 0,C 180,E1 31995.285,E2 31995.285} C_VEL
LIN {X 0,Y 696.424,Z 259.378,A -85,B 0,C 180,E1 31992.963,E2 31992.963} C_VEL
LIN {X 0,Y 698.188,Z 264.185,A -85,B 0,C 180,E1 31992.417,E2 31992.417} C_VEL
LIN {X 0,Y 705.14,Z 280.86,A -85,B 0,C 180,E1 31990.656,E2 31990.656} C_VEL
LIN {X 0,Y 705.319,Z 284.419,A -85,B 0,C 180,E1 31990.38,E2 31990.38} C_VEL
LIN {X 0,Y 705.412,Z 288.341,A -85,B 0,C 180,E1 31990.134,E2 31990.134} C_VEL
LIN {X 0,Y 709.335,Z 304.191,A -85,B 0,C 180,E1 31989.655,E2 31989.655} C_VEL
LIN {X 0,Y 707.434,Z 551.112,A -85,B 0,C 180,E1 31986.657,E2 31986.657} C_VEL
LIN {X 0,Y 706.162,Z 720.693,A -85,B 0,C 180,E1 31984.628,E2 31984.628} C_VEL
LIN {X 0,Y 705.738,Z 746.292,A -85,B 0,C 180,E1 31984.192,E2 31984.192} C_VEL
LIN {X 0,Y 705.067,Z 771.104,A -85,B 0,C 180,E1 31983.608,E2 31983.608} C_VEL
LIN {X 0,Y 704.457,Z 792.609,A -85,B 0,C 180,E1 31982.98,E2 31982.98} C_VEL
LIN {X 0,Y 703.71,Z 817.519,A -85,B 0,C 180,E1 31982.101,E2 31982.101} C_VEL
LIN {X 0,Y 702.871,Z 840.243,A -85,B 0,C 180,E1 31981.138,E2 31981.138} C_VEL
LIN {X 0,Y 702.069,Z 860.872,A -85,B 0,C 180,E1 31980.134,E2 31980.134} C_VEL
LIN {X 0,Y 701.118,Z 885.121,A -85,B 0,C 180,E1 31978.772,E2 31978.772} C_VEL
LIN {X 0,Y 700.352,Z 904.117,A -85,B 0,C 180,E1 31977.55,E2 31977.55} C_VEL
LIN {X 0,Y 699.533,Z 924.642,A -85,B 0,C 180,E1 31976.074,E2 31976.074} C_VEL
LIN {X 0,Y 698.786,Z 943.882,A -85,B 0,C 180,E1 31974.487,E2 31974.487} C_VEL
LIN {X 0,Y 698.146,Z 960.879,A -85,B 0,C 180,E1 31972.927,E2 31972.927} C_VEL
LIN {X 0,Y 697.546,Z 978.74,A -85,B 0,C 180,E1 31971.065,E2 31971.065} C_VEL
LIN {X 0,Y 697.079,Z 993.321,A -85,B 0,C 180,E1 31969.35,E2 31969.35} C_VEL
LIN {X 0,Y 696.667,Z 1008.698,A -85,B 0,C 180,E1 31967.283,E2 31967.283} C_VEL
LIN {X 0,Y 696.424,Z 1019.923,A -85,B 0,C 180,E1 31965.551,E2 31965.551} C_VEL
LIN {X 0,Y 696.218,Z 1030.872,A -85,B 0,C 180,E1 31963.623,E2 31963.623} C_VEL
LIN {X 0,Y 696.077,Z 1040.881,A -85,B 0,C 180,E1 31961.518,E2 31961.518} C_VEL
LIN {X 0,Y 695.969,Z 1047.877,A -85,B 0,C 180,E1 31959.76,E2 31959.76} C_VEL
LIN {X 0,Y 695.941,Z 1053.659,A -85,B 0,C 180,E1 31958.011,E2 31958.011} C_VEL
LIN {X 0,Y 695.908,Z 1059.209,A -85,B 0,C 180,E1 31955.855,E2 31955.855} C_VEL
LIN {X 0,Y 695.914,Z 1062.676,A -85,B 0,C 180,E1 31953.872,E2 31953.872} C_VEL
LIN {X 0,Y 695.906,Z 1064.573,A -85,B 0,C 180,E1 31952.141,E2 31952.141} C_VEL
LIN {X 0,Y 695.903,Z 1065.462,A -85,B 0,C 180,E1 31950.165,E2 31950.165} C_VEL
LIN {X 0,Y 695.908,Z 1064.707,A -85,B 0,C 180,E1 31948.024,E2 31948.024} C_VEL
LIN {X 0,Y 695.91,Z 1062.902,A -85,B 0,C 180,E1 31946.293,E2 31946.293} C_VEL
LIN {X 0,Y 695.903,Z 1060.007,A -85,B 0,C 180,E1 31944.559,E2 31944.559} C_VEL
LIN {X 0,Y 695.943,Z 1055.101,A -85,B 0,C 180,E1 31942.462,E2 31942.462} C_VEL
LIN {X 0,Y 695.969,Z 1048.487,A -85,B 0,C 180,E1 31940.407,E2 31940.407} C_VEL
LIN {X 0,Y 696.054,Z 1041.949,A -85,B 0,C 180,E1 31938.734,E2 31938.734} C_VEL
LIN {X 0,Y 696.175,Z 1033.84,A -85,B 0,C 180,E1 31936.968,E2 31936.968} C_VEL
LIN {X 0,Y 696.355,Z 1022.376,A -85,B 0,C 180,E1 31934.851,E2 31934.851} C_VEL
LIN {X 0,Y 696.611,Z 1011.023,A -85,B 0,C 180,E1 31933.06,E2 31933.06} C_VEL
LIN {X 0,Y 696.941,Z 998.716,A -85,B 0,C 180,E1 31931.341,E2 31931.341} C_VEL
LIN {X 0,Y 697.41,Z 982.426,A -85,B 0,C 180,E1 31929.348,E2 31929.348} C_VEL
LIN {X 0,Y 697.919,Z 967.571,A -85,B 0,C 180,E1 31927.746,E2 31927.746} C_VEL
LIN {X 0,Y 698.561,Z 949.631,A -85,B 0,C 180,E1 31926.015,E2 31926.015} C_VEL
LIN {X 0,Y 699.263,Z 931.298,A -85,B 0,C 180,E1 31924.46,E2 31924.46} C_VEL
LIN {X 0,Y 700.034,Z 911.923,A -85,B 0,C 180,E1 31922.986,E2 31922.986} C_VEL
LIN {X 0,Y 700.915,Z 890.236,A -85,B 0,C 180,E1 31921.545,E2 31921.545} C_VEL
LIN {X 0,Y 701.685,Z 871.02,A -85,B 0,C 180,E1 31920.412,E2 31920.412} C_VEL
LIN {X 0,Y 702.599,Z 847.208,A -85,B 0,C 180,E1 31919.181,E2 31919.181} C_VEL
LIN {X 0,Y 703.397,Z 825.422,A -85,B 0,C 180,E1 31918.219,E2 31918.219} C_VEL
LIN {X 0,Y 704.103,Z 804.973,A -85,B 0,C 180,E1 31917.438,E2 31917.438} C_VEL
LIN {X 0,Y 704.907,Z 779.499,A -85,B 0,C 180,E1 31916.62,E2 31916.62} C_VEL
LIN {X 0,Y 705.459,Z 755.371,A -85,B 0,C 180,E1 31916.006,E2 31916.006} C_VEL
LIN {X 0,Y 705.911,Z 733.179,A -85,B 0,C 180,E1 31915.565,E2 31915.565} C_VEL
LIN {X 0,Y 706.36,Z 702.917,A -85,B 0,C 180,E1 31915.142,E2 31915.142} C_VEL
LIN {X 0,Y 708.099,Z 461.328,A -85,B 0,C 180,E1 31912.263,E2 31912.263} C_VEL
LIN {X 0,Y 709.19,Z 302.95,A -85,B 0,C 180,E1 31910.319,E2 31910.319} C_VEL
LIN {X 0,Y 705.28,Z 287.479,A -85,B 0,C 180,E1 31909.83,E2 31909.83} C_VEL
LIN {X 0,Y 705.383,Z 281.53,A -85,B 0,C 180,E1 31909.411,E2 31909.411} C_VEL
LIN {X 0,Y 699.092,Z 266.226,A -85,B 0,C 180,E1 31907.807,E2 31907.807} C_VEL
LIN {X 0,Y 696.448,Z 259.531,A -85,B 0,C 180,E1 31907.072,E2 31907.072} C_VEL
LIN {X 0,Y 696.328,Z 259.225,A -85,B 0,C 180,E1 31905.973,E2 31905.973} C_VEL
LIN {X 0,Y 696.404,Z 259.217,A -85,B 0,C 180,E1 31903.113,E2 31903.113} C_VEL
LIN {X 0,Y 696.331,Z 259.238,A -85,B 0,C 180,E1 31900.189,E2 31900.189} C_VEL
LIN {X 0,Y 696.341,Z 259.229,A -85,B 0,C 180,E1 31897.609,E2 31897.609} C_VEL
LIN {X 0,Y 696.368,Z 259.22,A -85,B 0,C 180,E1 31894.553,E2 31894.553} C_VEL
LIN {X 0,Y 696.326,Z 259.238,A -85,B 0,C 180,E1 31891.9,E2 31891.9} C_VEL
LIN {X 0,Y 696.371,Z 259.225,A -85,B 0,C 180,E1 31889.191,E2 31889.191} C_VEL
LIN {X 0,Y 696.343,Z 259.239,A -85,B 0,C 180,E1 31886.157,E2 31886.157} C_VEL
LIN {X 0,Y 696.328,Z 259.232,A -85,B 0,C 180,E1 31883.618,E2 31883.618} C_VEL
LIN {X 0,Y 696.406,Z 259.233,A -85,B 0,C 180,E1 31880.771,E2 31880.771} C_VEL
LIN {X 0,Y 696.331,Z 259.236,A -85,B 0,C 180,E1 31877.82,E2 31877.82} C_VEL
LIN {X 0,Y 696.343,Z 259.234,A -85,B 0,C 180,E1 31875.219,E2 31875.219} C_VEL
LIN {X 0,Y 696.359,Z 259.238,A -85,B 0,C 180,E1 31872.101,E2 31872.101} C_VEL
LIN {X 0,Y 696.327,Z 259.234,A -85,B 0,C 180,E1 31869.429,E2 31869.429} C_VEL
LIN {X 0,Y 696.406,Z 259.231,A -85,B 0,C 180,E1 31866.596,E2 31866.596} C_VEL
LIN {X 0,Y 696.33,Z 259.235,A -85,B 0,C 180,E1 31863.622,E2 31863.622} C_VEL
LIN {X 0,Y 696.336,Z 259.234,A -85,B 0,C 180,E1 31861.07,E2 31861.07} C_VEL
LIN {X 0,Y 696.391,Z 259.24,A -85,B 0,C 180,E1 31858.108,E2 31858.108} C_VEL
LIN {X 0,Y 696.325,Z 259.232,A -85,B 0,C 180,E1 31855.305,E2 31855.305} C_VEL
LIN {X 0,Y 696.361,Z 259.234,A -85,B 0,C 180,E1 31852.658,E2 31852.658} C_VEL
LIN {X 0,Y 696.343,Z 259.238,A -85,B 0,C 180,E1 31849.576,E2 31849.576} C_VEL
LIN {X 0,Y 696.328,Z 259.229,A -85,B 0,C 180,E1 31846.971,E2 31846.971} C_VEL
LIN {X 0,Y 696.408,Z 259.236,A -85,B 0,C 180,E1 31844.084,E2 31844.084} C_VEL
LIN {X 0,Y 696.329,Z 259.238,A -85,B 0,C 180,E1 31841.237,E2 31841.237} C_VEL
LIN {X 0,Y 696.335,Z 259.23,A -85,B 0,C 180,E1 31838.697,E2 31838.697} C_VEL
LIN {X 0,Y 696.392,Z 259.228,A -85,B 0,C 180,E1 31835.746,E2 31835.746} C_VEL
LIN {X 0,Y 696.339,Z 259.226,A -85,B 0,C 180,E1 31835.32,E2 31835.32} C_VEL
LIN {X 0,Y 695.305,Z 259.352,A -85,B 0,C 180,E1 31834.686,E2 31834.686} C_VEL
LIN {X 0,Y 688.902,Z 260.143,A -85,B 0,C 180,E1 31832.91,E2 31832.91} C_VEL
LIN {X 0,Y 688.406,Z 260.206,A -85,B 0,C 180,E1 31832.448,E2 31832.448} C_VEL
LIN {X 0,Y 688.408,Z 260.223,A -85,B 0,C 180,E1 31829.3,E2 31829.3} C_VEL
LIN {X 0,Y 688.385,Z 260.201,A -85,B 0,C 180,E1 31826.698,E2 31826.698} C_VEL
LIN {X 0,Y 688.47,Z 260.225,A -85,B 0,C 180,E1 31823.765,E2 31823.765} C_VEL
LIN {X 0,Y 688.39,Z 260.229,A -85,B 0,C 180,E1 31820.862,E2 31820.862} C_VEL
LIN {X 0,Y 688.399,Z 260.222,A -85,B 0,C 180,E1 31818.294,E2 31818.294} C_VEL
LIN {X 0,Y 688.425,Z 260.227,A -85,B 0,C 180,E1 31815.216,E2 31815.216} C_VEL
LIN {X 0,Y 688.386,Z 260.232,A -85,B 0,C 180,E1 31812.572,E2 31812.572} C_VEL
LIN {X 0,Y 688.423,Z 260.216,A -85,B 0,C 180,E1 31809.924,E2 31809.924} C_VEL
LIN {X 0,Y 688.538,Z 260.706,A -85,B 0,C 180,E1 31809.654,E2 31809.654} C_VEL
LIN {X 0,Y 695.707,Z 278.104,A -85,B 0,C 180,E1 31807.77,E2 31807.77} C_VEL
LIN {X 0,Y 700.799,Z 286.954,A -85,B 0,C 180,E1 31807.287,E2 31807.287} C_VEL
LIN {X 0,Y 703.149,Z 296.684,A -85,B 0,C 180,E1 31806.997,E2 31806.997} C_VEL
LIN {X 0,Y 700.987,Z 544.134,A -85,B 0,C 180,E1 31803.967,E2 31803.967} C_VEL
LIN {X 0,Y 699.568,Z 710.77,A -85,B 0,C 180,E1 31801.955,E2 31801.955} C_VEL
LIN {X 0,Y 699.077,Z 736.646,A -85,B 0,C 180,E1 31801.51,E2 31801.51} C_VEL
LIN {X 0,Y 698.353,Z 761.077,A -85,B 0,C 180,E1 31800.931,E2 31800.931} C_VEL
LIN {X 0,Y 697.654,Z 782.651,A -85,B 0,C 180,E1 31800.297,E2 31800.297} C_VEL
LIN {X 0,Y 696.772,Z 808.039,A -85,B 0,C 180,E1 31799.392,E2 31799.392} C_VEL
LIN {X 0,Y 695.88,Z 829.862,A -85,B 0,C 180,E1 31798.46,E2 31798.46} C_VEL
LIN {X 0,Y 695.032,Z 849.455,A -85,B 0,C 180,E1 31797.503,E2 31797.503} C_VEL
LIN {X 0,Y 693.977,Z 872.696,A -85,B 0,C 180,E1 31796.206,E2 31796.206} C_VEL
LIN {X 0,Y 693.034,Z 893.425,A -85,B 0,C 180,E1 31794.87,E2 31794.87} C_VEL
LIN {X 0,Y 692.146,Z 912.928,A -85,B 0,C 180,E1 31793.46,E2 31793.46} C_VEL
LIN {X 0,Y 691.249,Z 932.809,A -85,B 0,C 180,E1 31791.823,E2 31791.823} C_VEL
LIN {X 0,Y 690.578,Z 948.969,A -85,B 0,C 180,E1 31790.334,E2 31790.334} C_VEL
LIN {X 0,Y 689.833,Z 967.404,A -85,B 0,C 180,E1 31788.42,E2 31788.42} C_VEL
LIN {X 0,Y 689.314,Z 982.057,A -85,B 0,C 180,E1 31786.691,E2 31786.691} C_VEL
LIN {X 0,Y 688.859,Z 996.874,A -85,B 0,C 180,E1 31784.715,E2 31784.715} C_VEL
LIN {X 0,Y 688.518,Z 1009.031,A -85,B 0,C 180,E1 31782.838,E2 31782.838} C_VEL
LIN {X 0,Y 688.298,Z 1019.174,A -85,B 0,C 180,E1 31781.055,E2 31781.055} C_VEL
LIN {X 0,Y 688.105,Z 1029.471,A -85,B 0,C 180,E1 31778.945,E2 31778.945} C_VEL
LIN {X 0,Y 688.004,Z 1037.219,A -85,B 0,C 180,E1 31777.012,E2 31777.012} C_VEL
LIN {X 0,Y 687.95,Z 1042.817,A -85,B 0,C 180,E1 31775.337,E2 31775.337} C_VEL
LIN {X 0,Y 687.93,Z 1047.568,A -85,B 0,C 180,E1 31773.583,E2 31773.583} C_VEL
LIN {X 0,Y 687.896,Z 1051.823,A -85,B 0,C 180,E1 31771.499,E2 31771.499} C_VEL
LIN {X 0,Y 687.906,Z 1054.334,A -85,B 0,C 180,E1 31769.417,E2 31769.417} C_VEL
LIN {X 0,Y 687.893,Z 1055.338,A -85,B 0,C 180,E1 31767.584,E2 31767.584} C_VEL
LIN {X 0,Y 687.905,Z 1055.137,A -85,B 0,C 180,E1 31765.582,E2 31765.582} C_VEL
LIN {X 0,Y 687.907,Z 1053.175,A -85,B 0,C 180,E1 31763.406,E2 31763.406} C_VEL
LIN {X 0,Y 687.91,Z 1050.373,A -85,B 0,C 180,E1 31761.642,E2 31761.642} C_VEL
LIN {X 0,Y 687.938,Z 1046.444,A -85,B 0,C 180,E1 31759.871,E2 31759.871} C_VEL
LIN {X 0,Y 687.991,Z 1040.285,A -85,B 0,C 180,E1 31757.749,E2 31757.749} C_VEL
LIN {X 0,Y 688.069,Z 1032.542,A -85,B 0,C 180,E1 31755.698,E2 31755.698} C_VEL
LIN {X 0,Y 688.196,Z 1024.826,A -85,B 0,C 180,E1 31753.975,E2 31753.975} C_VEL
LIN {X 0,Y 688.392,Z 1014.431,A -85,B 0,C 180,E1 31751.978,E2 31751.978} C_VEL
LIN {X 0,Y 688.7,Z 1001.884,A -85,B 0,C 180,E1 31749.943,E2 31749.943} C_VEL
LIN {X 0,Y 689.071,Z 989.584,A -85,B 0,C 180,E1 31748.194,E2 31748.194} C_VEL
LIN {X 0,Y 689.603,Z 973.608,A -85,B 0,C 180,E1 31746.195,E2 31746.195} C_VEL
LIN {X 0,Y 690.199,Z 958.107,A -85,B 0,C 180,E1 31744.495,E2 31744.495} C_VEL
LIN {X 0,Y 690.951,Z 940.215,A -85,B 0,C 180,E1 31742.741,E2 31742.741} C_VEL
LIN {X 0,Y 691.74,Z 921.804,A -85,B 0,C 180,E1 31741.159,E2 31741.159} C_VEL
LIN {X 0,Y 692.559,Z 903.472,A -85,B 0,C 180,E1 31739.744,E2 31739.744} C_VEL
LIN {X 0,Y 693.588,Z 881.478,A -85,B 0,C 180,E1 31738.252,E2 31738.252} C_VEL
LIN {X 0,Y 694.441,Z 862.67,A -85,B 0,C 180,E1 31737.124,E2 31737.124} C_VEL
LIN {X 0,Y 695.388,Z 841.323,A -85,B 0,C 180,E1 31735.99,E2 31735.99} C_VEL
LIN {X 0,Y 696.403,Z 816.765,A -85,B 0,C 180,E1 31734.876,E2 31734.876} C_VEL
LIN {X 0,Y 697.194,Z 796.446,A -85,B 0,C 180,E1 31734.086,E2 31734.086} C_VEL
LIN {X 0,Y 698.01,Z 773.905,A -85,B 0,C 180,E1 31733.34,E2 31733.34} C_VEL
LIN {X 0,Y 698.741,Z 747.557,A -85,B 0,C 180,E1 31732.641,E2 31732.641} C_VEL
LIN {X 0,Y 699.242,Z 725.361,A -85,B 0,C 180,E1 31732.187,E2 31732.187} C_VEL
LIN {X 0,Y 699.72,Z 700.407,A -85,B 0,C 180,E1 31731.812,E2 31731.812} C_VEL
LIN {X 0,Y 701.724,Z 456.966,A -85,B 0,C 180,E1 31728.886,E2 31728.886} C_VEL
LIN {X 0,Y 702.985,Z 295.261,A -85,B 0,C 180,E1 31726.883,E2 31726.883} C_VEL
LIN {X 0,Y 700.288,Z 285.71,A -85,B 0,C 180,E1 31726.572,E2 31726.572} C_VEL
LIN {X 0,Y 695.604,Z 277.895,A -85,B 0,C 180,E1 31726.127,E2 31726.127} C_VEL
LIN {X 0,Y 688.495,Z 260.482,A -85,B 0,C 180,E1 31724.22,E2 31724.22} C_VEL
LIN {X 0,Y 688.388,Z 260.231,A -85,B 0,C 180,E1 31721.454,E2 31721.454} C_VEL
LIN {X 0,Y 688.407,Z 260.231,A -85,B 0,C 180,E1 31718.864,E2 31718.864} C_VEL
LIN {X 0,Y 688.412,Z 260.226,A -85,B 0,C 180,E1 31715.716,E2 31715.716} C_VEL
LIN {X 0,Y 688.388,Z 260.225,A -85,B 0,C 180,E1 31713.103,E2 31713.103} C_VEL
LIN {X 0,Y 688.468,Z 260.213,A -85,B 0,C 180,E1 31710.216,E2 31710.216} C_VEL
LIN {X 0,Y 688.392,Z 260.222,A -85,B 0,C 180,E1 31707.322,E2 31707.322} C_VEL
LIN {X 0,Y 688.396,Z 260.213,A -85,B 0,C 180,E1 31704.729,E2 31704.729} C_VEL
LIN {X 0,Y 688.444,Z 260.215,A -85,B 0,C 180,E1 31701.738,E2 31701.738} C_VEL
LIN {X 0,Y 688.387,Z 260.214,A -85,B 0,C 180,E1 31698.988,E2 31698.988} C_VEL
LIN {X 0,Y 688.435,Z 260.229,A -85,B 0,C 180,E1 31696.253,E2 31696.253} C_VEL
LIN {X 0,Y 688.403,Z 260.208,A -85,B 0,C 180,E1 31693.267,E2 31693.267} C_VEL
LIN {X 0,Y 688.391,Z 260.226,A -85,B 0,C 180,E1 31690.63,E2 31690.63} C_VEL
LIN {X 0,Y 688.467,Z 260.196,A -85,B 0,C 180,E1 31687.679,E2 31687.679} C_VEL
LIN {X 0,Y 688.388,Z 260.221,A -85,B 0,C 180,E1 31684.833,E2 31684.833} C_VEL
LIN {X 0,Y 688.416,Z 260.227,A -85,B 0,C 180,E1 31682.164,E2 31682.164} C_VEL
LIN {X 0,Y 688.408,Z 260.213,A -85,B 0,C 180,E1 31679.085,E2 31679.085} C_VEL
LIN {X 0,Y 688.389,Z 260.226,A -85,B 0,C 180,E1 31676.502,E2 31676.502} C_VEL
LIN {X 0,Y 688.462,Z 260.2,A -85,B 0,C 180,E1 31673.663,E2 31673.663} C_VEL
LIN {X 0,Y 688.393,Z 260.221,A -85,B 0,C 180,E1 31670.722,E2 31670.722} C_VEL
LIN {X 0,Y 688.401,Z 260.224,A -85,B 0,C 180,E1 31668.097,E2 31668.097} C_VEL
LIN {X 0,Y 688.425,Z 260.216,A -85,B 0,C 180,E1 31664.986,E2 31664.986} C_VEL
LIN {X 0,Y 688.389,Z 260.225,A -85,B 0,C 180,E1 31662.328,E2 31662.328} C_VEL
LIN {X 0,Y 688.452,Z 260.203,A -85,B 0,C 180,E1 31659.511,E2 31659.511} C_VEL
LIN {X 0,Y 688.397,Z 260.225,A -85,B 0,C 180,E1 31656.548,E2 31656.548} C_VEL
LIN {X 0,Y 688.395,Z 260.224,A -85,B 0,C 180,E1 31653.982,E2 31653.982} C_VEL
LIN {X 0,Y 688.458,Z 260.224,A -85,B 0,C 180,E1 31650.982,E2 31650.982} C_VEL
LIN {X 0,Y 688.387,Z 260.216,A -85,B 0,C 180,E1 31648.179,E2 31648.179} C_VEL
LIN {X 0,Y 688.432,Z 260.218,A -85,B 0,C 180,E1 31645.438,E2 31645.438} C_VEL
LIN {X 0,Y 688.401,Z 260.205,A -85,B 0,C 180,E1 31642.407,E2 31642.407} C_VEL
LIN {X 0,Y 688.392,Z 260.229,A -85,B 0,C 180,E1 31639.819,E2 31639.819} C_VEL
LIN {X 0,Y 688.466,Z 260.221,A -85,B 0,C 180,E1 31636.93,E2 31636.93} C_VEL
LIN {X 0,Y 688.389,Z 260.215,A -85,B 0,C 180,E1 31634.028,E2 31634.028} C_VEL
LIN {X 0,Y 688.442,Z 260.478,A -85,B 0,C 180,E1 31633.471,E2 31633.471} C_VEL
LIN {X 0,Y 698.327,Z 284.419,A -85,B 0,C 180,E1 31630.87,E2 31630.87} C_VEL
LIN {X 0,Y 698.579,Z 286.669,A -85,B 0,C 180,E1 31630.684,E2 31630.684} C_VEL
LIN {X 0,Y 698.954,Z 289.35,A -85,B 0,C 180,E1 31630.561,E2 31630.561} C_VEL
LIN {X 0,Y 703.151,Z 306.217,A -85,B 0,C 180,E1 31630.048,E2 31630.048} C_VEL
LIN {X 0,Y 701,Z 552.511,A -85,B 0,C 180,E1 31627.032,E2 31627.032} C_VEL
LIN {X 0,Y 699.569,Z 720.601,A -85,B 0,C 180,E1 31625.003,E2 31625.003} C_VEL
LIN {X 0,Y 699.093,Z 746.244,A -85,B 0,C 180,E1 31624.564,E2 31624.564} C_VEL
LIN {X 0,Y 698.355,Z 771.001,A -85,B 0,C 180,E1 31623.978,E2 31623.978} C_VEL
LIN {X 0,Y 697.656,Z 792.664,A -85,B 0,C 180,E1 31623.342,E2 31623.342} C_VEL
LIN {X 0,Y 696.749,Z 818.645,A -85,B 0,C 180,E1 31622.412,E2 31622.412} C_VEL
LIN {X 0,Y 695.861,Z 840.239,A -85,B 0,C 180,E1 31621.488,E2 31621.488} C_VEL
LIN {X 0,Y 695.006,Z 859.986,A -85,B 0,C 180,E1 31620.521,E2 31620.521} C_VEL
LIN {X 0,Y 693.931,Z 883.65,A -85,B 0,C 180,E1 31619.192,E2 31619.192} C_VEL
LIN {X 0,Y 693.033,Z 903.416,A -85,B 0,C 180,E1 31617.916,E2 31617.916} C_VEL
LIN {X 0,Y 692.15,Z 922.833,A -85,B 0,C 180,E1 31616.512,E2 31616.512} C_VEL
LIN {X 0,Y 691.26,Z 942.533,A -85,B 0,C 180,E1 31614.893,E2 31614.893} C_VEL
LIN {X 0,Y 690.574,Z 959.026,A -85,B 0,C 180,E1 31613.374,E2 31613.374} C_VEL
LIN {X 0,Y 689.82,Z 977.764,A -85,B 0,C 180,E1 31611.424,E2 31611.424} C_VEL
LIN {X 0,Y 689.306,Z 992.29,A -85,B 0,C 180,E1 31609.707,E2 31609.707} C_VEL
LIN {X 0,Y 688.855,Z 1006.958,A -85,B 0,C 180,E1 31607.747,E2 31607.747} C_VEL
LIN {X 0,Y 688.513,Z 1019.262,A -85,B 0,C 180,E1 31605.844,E2 31605.844} C_VEL
LIN {X 0,Y 688.288,Z 1029.494,A -85,B 0,C 180,E1 31604.04,E2 31604.04} C_VEL
LIN {X 0,Y 688.103,Z 1040.17,A -85,B 0,C 180,E1 31601.823,E2 31601.823} C_VEL
LIN {X 0,Y 687.993,Z 1047.573,A -85,B 0,C 180,E1 31599.959,E2 31599.959} C_VEL
LIN {X 0,Y 687.955,Z 1053.149,A -85,B 0,C 180,E1 31598.273,E2 31598.273} C_VEL
LIN {X 0,Y 687.927,Z 1058.273,A -85,B 0,C 180,E1 31596.342,E2 31596.342} C_VEL
LIN {X 0,Y 687.913,Z 1062.451,A -85,B 0,C 180,E1 31594.084,E2 31594.084} C_VEL
LIN {X 0,Y 687.903,Z 1064.439,A -85,B 0,C 180,E1 31592.333,E2 31592.333} C_VEL
LIN {X 0,Y 687.892,Z 1065.35,A -85,B 0,C 180,E1 31590.583,E2 31590.583} C_VEL
LIN {X 0,Y 687.896,Z 1065.1,A -85,B 0,C 180,E1 31588.501,E2 31588.501} C_VEL
LIN {X 0,Y 687.905,Z 1063.128,A -85,B 0,C 180,E1 31586.417,E2 31586.417} C_VEL
LIN {X 0,Y 687.909,Z 1060.325,A -85,B 0,C 180,E1 31584.662,E2 31584.662} C_VEL
LIN {X 0,Y 687.941,Z 1056.413,A -85,B 0,C 180,E1 31582.903,E2 31582.903} C_VEL
LIN {X 0,Y 687.992,Z 1050.308,A -85,B 0,C 180,E1 31580.801,E2 31580.801} C_VEL
LIN {X 0,Y 688.065,Z 1042.662,A -85,B 0,C 180,E1 31578.771,E2 31578.771} C_VEL
LIN {X 0,Y 688.199,Z 1034.659,A -85,B 0,C 180,E1 31576.985,E2 31576.985} C_VEL
LIN {X 0,Y 688.401,Z 1023.918,A -85,B 0,C 180,E1 31574.93,E2 31574.93} C_VEL
LIN {X 0,Y 688.707,Z 1011.605,A -85,B 0,C 180,E1 31572.946,E2 31572.946} C_VEL
LIN {X 0,Y 689.081,Z 999.361,A -85,B 0,C 180,E1 31571.208,E2 31571.208} C_VEL
LIN {X 0,Y 689.62,Z 983.194,A -85,B 0,C 180,E1 31569.193,E2 31569.193} C_VEL
LIN {X 0,Y 690.206,Z 967.867,A -85,B 0,C 180,E1 31567.515,E2 31567.515} C_VEL
LIN {X 0,Y 690.976,Z 949.63,A -85,B 0,C 180,E1 31565.735,E2 31565.735} C_VEL
LIN {X 0,Y 691.762,Z 931.274,A -85,B 0,C 180,E1 31564.161,E2 31564.161} C_VEL
LIN {X 0,Y 692.671,Z 911.312,A -85,B 0,C 180,E1 31562.628,E2 31562.628} C_VEL
LIN {X 0,Y 693.646,Z 890.178,A -85,B 0,C 180,E1 31561.215,E2 31561.215} C_VEL
LIN {X 0,Y 694.511,Z 871.057,A -85,B 0,C 180,E1 31560.078,E2 31560.078} C_VEL
LIN {X 0,Y 695.559,Z 847.212,A -85,B 0,C 180,E1 31558.835,E2 31558.835} C_VEL
LIN {X 0,Y 696.464,Z 825.427,A -85,B 0,C 180,E1 31557.865,E2 31557.865} C_VEL
LIN {X 0,Y 697.257,Z 804.97,A -85,B 0,C 180,E1 31557.078,E2 31557.078} C_VEL
LIN {X 0,Y 698.141,Z 779.942,A -85,B 0,C 180,E1 31556.266,E2 31556.266} C_VEL
LIN {X 0,Y 698.773,Z 755.45,A -85,B 0,C 180,E1 31555.638,E2 31555.638} C_VEL
LIN {X 0,Y 699.299,Z 733.178,A -85,B 0,C 180,E1 31555.193,E2 31555.193} C_VEL
LIN {X 0,Y 699.791,Z 702.917,A -85,B 0,C 180,E1 31554.766,E2 31554.766} C_VEL
LIN {X 0,Y 701.762,Z 461.755,A -85,B 0,C 180,E1 31551.867,E2 31551.867} C_VEL
LIN {X 0,Y 703.005,Z 304.941,A -85,B 0,C 180,E1 31549.925,E2 31549.925} C_VEL
LIN {X 0,Y 698.597,Z 287.462,A -85,B 0,C 180,E1 31549.366,E2 31549.366} C_VEL
LIN {X 0,Y 698.628,Z 285.213,A -85,B 0,C 180,E1 31549.211,E2 31549.211} C_VEL
LIN {X 0,Y 690.836,Z 266.473,A -85,B 0,C 180,E1 31547.207,E2 31547.207} C_VEL
LIN {X 0,Y 688.43,Z 260.408,A -85,B 0,C 180,E1 31546.51,E2 31546.51} C_VEL
LIN {X 0,Y 688.392,Z 260.23,A -85,B 0,C 180,E1 31543.971,E2 31543.971} C_VEL
LIN {X 0,Y 688.467,Z 260.221,A -85,B 0,C 180,E1 31541.031,E2 31541.031} C_VEL
LIN {X 0,Y 688.39,Z 260.217,A -85,B 0,C 180,E1 31538.121,E2 31538.121} C_VEL
LIN {X 0,Y 688.408,Z 260.225,A -85,B 0,C 180,E1 31535.52,E2 31535.52} C_VEL
LIN {X 0,Y 688.418,Z 260.227,A -85,B 0,C 180,E1 31532.409,E2 31532.409} C_VEL
LIN {X 0,Y 688.389,Z 260.218,A -85,B 0,C 180,E1 31529.786,E2 31529.786} C_VEL
LIN {X 0,Y 688.447,Z 260.212,A -85,B 0,C 180,E1 31527.039,E2 31527.039} C_VEL
LIN {X 0,Y 688.4,Z 260.222,A -85,B 0,C 180,E1 31524.089,E2 31524.089} C_VEL
LIN {X 0,Y 688.39,Z 260.225,A -85,B 0,C 180,E1 31521.561,E2 31521.561} C_VEL
LIN {X 0,Y 688.468,Z 260.223,A -85,B 0,C 180,E1 31518.634,E2 31518.634} C_VEL
LIN {X 0,Y 688.39,Z 260.225,A -85,B 0,C 180,E1 31515.761,E2 31515.761} C_VEL
LIN {X 0,Y 688.403,Z 260.222,A -85,B 0,C 180,E1 31513.182,E2 31513.182} C_VEL
LIN {X 0,Y 688.417,Z 260.226,A -85,B 0,C 180,E1 31510.038,E2 31510.038} C_VEL
LIN {X 0,Y 688.387,Z 260.224,A -85,B 0,C 180,E1 31507.428,E2 31507.428} C_VEL
LIN {X 0,Y 688.448,Z 260.221,A -85,B 0,C 180,E1 31504.665,E2 31504.665} C_VEL
LIN {X 0,Y 688.397,Z 260.226,A -85,B 0,C 180,E1 31501.665,E2 31501.665} C_VEL
LIN {X 0,Y 688.393,Z 260.221,A -85,B 0,C 180,E1 31499.085,E2 31499.085} C_VEL
LIN {X 0,Y 688.451,Z 260.22,A -85,B 0,C 180,E1 31496.086,E2 31496.086} C_VEL
LIN {X 0,Y 688.387,Z 260.226,A -85,B 0,C 180,E1 31493.327,E2 31493.327} C_VEL
LIN {X 0,Y 688.41,Z 260.217,A -85,B 0,C 180,E1 31490.722,E2 31490.722} C_VEL
LIN {X 0,Y 688.407,Z 260.22,A -85,B 0,C 180,E1 31487.586,E2 31487.586} C_VEL
LIN {X 0,Y 688.388,Z 260.226,A -85,B 0,C 180,E1 31484.997,E2 31484.997} C_VEL
LIN {X 0,Y 688.465,Z 260.216,A -85,B 0,C 180,E1 31482.155,E2 31482.155} C_VEL
LIN {X 0,Y 688.392,Z 260.22,A -85,B 0,C 180,E1 31479.243,E2 31479.243} C_VEL
LIN {X 0,Y 688.393,Z 260.225,A -85,B 0,C 180,E1 31476.729,E2 31476.729} C_VEL
LIN {X 0,Y 688.457,Z 260.196,A -85,B 0,C 180,E1 31473.799,E2 31473.799} C_VEL
LIN {X 0,Y 688.406,Z 260.206,A -85,B 0,C 180,E1 31472.448,E2 31472.448} C_VEL
LIN {X 0,Y 687.476,Z 260.333,A -85,B 0,C 180,E1 31471.807,E2 31471.807} C_VEL
LIN {X 0,Y 680.987,Z 261.158,A -85,B 0,C 180,E1 31469.965,E2 31469.965} C_VEL
LIN {X 0,Y 680.498,Z 261.213,A -85,B 0,C 180,E1 31469.544,E2 31469.544} C_VEL
LIN {X 0,Y 680.444,Z 261.187,A -85,B 0,C 180,E1 31466.863,E2 31466.863} C_VEL
LIN {X 0,Y 680.493,Z 261.212,A -85,B 0,C 180,E1 31464.107,E2 31464.107} C_VEL
LIN {X 0,Y 680.459,Z 261.219,A -85,B 0,C 180,E1 31461.016,E2 31461.016} C_VEL
LIN {X 0,Y 680.455,Z 261.211,A -85,B 0,C 180,E1 31458.412,E2 31458.412} C_VEL
LIN {X 0,Y 680.508,Z 261.209,A -85,B 0,C 180,E1 31455.385,E2 31455.385} C_VEL
LIN {X 0,Y 680.447,Z 261.219,A -85,B 0,C 180,E1 31452.591,E2 31452.591} C_VEL
LIN {X 0,Y 680.49,Z 261.452,A -85,B 0,C 180,E1 31450.249,E2 31450.249} C_VEL
LIN {X 0,Y 686.733,Z 276.742,A -85,B 0,C 180,E1 31448.5,E2 31448.5} C_VEL
LIN {X 0,Y 688.2,Z 279.451,A -85,B 0,C 180,E1 31448.285,E2 31448.285} C_VEL
LIN {X 0,Y 695.285,Z 291.32,A -85,B 0,C 180,E1 31447.615,E2 31447.615} C_VEL
LIN {X 0,Y 696.998,Z 298.77,A -85,B 0,C 180,E1 31447.395,E2 31447.395} C_VEL
LIN {X 0,Y 694.58,Z 545.646,A -85,B 0,C 180,E1 31444.348,E2 31444.348} C_VEL
LIN {X 0,Y 693.004,Z 710.802,A -85,B 0,C 180,E1 31442.336,E2 31442.336} C_VEL
LIN {X 0,Y 692.453,Z 736.788,A -85,B 0,C 180,E1 31441.885,E2 31441.885} C_VEL
LIN {X 0,Y 691.669,Z 761.008,A -85,B 0,C 180,E1 31441.307,E2 31441.307} C_VEL
LIN {X 0,Y 690.902,Z 782.457,A -85,B 0,C 180,E1 31440.673,E2 31440.673} C_VEL
LIN {X 0,Y 689.883,Z 808.106,A -85,B 0,C 180,E1 31439.753,E2 31439.753} C_VEL
LIN {X 0,Y 688.888,Z 830.039,A -85,B 0,C 180,E1 31438.808,E2 31438.808} C_VEL
LIN {X 0,Y 687.96,Z 849.35,A -85,B 0,C 180,E1 31437.857,E2 31437.857} C_VEL
LIN {X 0,Y 686.777,Z 872.606,A -85,B 0,C 180,E1 31436.549,E2 31436.549} C_VEL
LIN {X 0,Y 685.71,Z 893.348,A -85,B 0,C 180,E1 31435.2,E2 31435.2} C_VEL
LIN {X 0,Y 684.716,Z 912.953,A -85,B 0,C 180,E1 31433.768,E2 31433.768} C_VEL
LIN {X 0,Y 683.696,Z 932.752,A -85,B 0,C 180,E1 31432.122,E2 31432.122} C_VEL
LIN {X 0,Y 682.957,Z 948.462,A -85,B 0,C 180,E1 31430.661,E2 31430.661} C_VEL
LIN {X 0,Y 682.146,Z 966.215,A -85,B 0,C 180,E1 31428.813,E2 31428.813} C_VEL
LIN {X 0,Y 681.537,Z 981.668,A -85,B 0,C 180,E1 31426.975,E2 31426.975} C_VEL
LIN {X 0,Y 681.002,Z 996.555,A -85,B 0,C 180,E1 31424.976,E2 31424.976} C_VEL
LIN {X 0,Y 680.596,Z 1009.258,A -85,B 0,C 180,E1 31422.99,E2 31422.99} C_VEL
LIN {X 0,Y 680.356,Z 1019.37,A -85,B 0,C 180,E1 31421.186,E2 31421.186} C_VEL
LIN {X 0,Y 680.125,Z 1029.977,A -85,B 0,C 180,E1 31418.965,E2 31418.965} C_VEL
LIN {X 0,Y 680.023,Z 1037.35,A -85,B 0,C 180,E1 31417.095,E2 31417.095} C_VEL
LIN {X 0,Y 679.956,Z 1043.18,A -85,B 0,C 180,E1 31415.316,E2 31415.316} C_VEL
LIN {X 0,Y 679.928,Z 1048.272,A -85,B 0,C 180,E1 31413.372,E2 31413.372} C_VEL
LIN {X 0,Y 679.912,Z 1052.44,A -85,B 0,C 180,E1 31411.095,E2 31411.095} C_VEL
LIN {X 0,Y 679.901,Z 1054.43,A -85,B 0,C 180,E1 31409.326,E2 31409.326} C_VEL
LIN {X 0,Y 679.892,Z 1055.347,A -85,B 0,C 180,E1 31407.556,E2 31407.556} C_VEL
LIN {X 0,Y 679.897,Z 1055.103,A -85,B 0,C 180,E1 31405.445,E2 31405.445} C_VEL
LIN {X 0,Y 679.908,Z 1053.127,A -85,B 0,C 180,E1 31403.328,E2 31403.328} C_VEL
LIN {X 0,Y 679.906,Z 1050.305,A -85,B 0,C 180,E1 31401.543,E2 31401.543} C_VEL
LIN {X 0,Y 679.945,Z 1046.355,A -85,B 0,C 180,E1 31399.75,E2 31399.75} C_VEL
LIN {X 0,Y 679.997,Z 1040.152,A -85,B 0,C 180,E1 31397.603,E2 31397.603} C_VEL
LIN {X 0,Y 680.094,Z 1032.748,A -85,B 0,C 180,E1 31395.613,E2 31395.613} C_VEL
LIN {X 0,Y 680.236,Z 1025.062,A -85,B 0,C 180,E1 31393.87,E2 31393.87} C_VEL
LIN {X 0,Y 680.441,Z 1015.169,A -85,B 0,C 180,E1 31391.937,E2 31391.937} C_VEL
LIN {X 0,Y 680.802,Z 1002.287,A -85,B 0,C 180,E1 31389.801,E2 31389.801} C_VEL
LIN {X 0,Y 681.227,Z 989.953,A -85,B 0,C 180,E1 31388.02,E2 31388.02} C_VEL
LIN {X 0,Y 681.827,Z 974.158,A -85,B 0,C 180,E1 31386.011,E2 31386.011} C_VEL
LIN {X 0,Y 682.481,Z 958.739,A -85,B 0,C 180,E1 31384.294,E2 31384.294} C_VEL
LIN {X 0,Y 683.35,Z 940.789,A -85,B 0,C 180,E1 31382.507,E2 31382.507} C_VEL
LIN {X 0,Y 684.248,Z 921.802,A -85,B 0,C 180,E1 31380.855,E2 31380.855} C_VEL
LIN {X 0,Y 685.206,Z 902.919,A -85,B 0,C 180,E1 31379.384,E2 31379.384} C_VEL
LIN {X 0,Y 686.364,Z 880.823,A -85,B 0,C 180,E1 31377.878,E2 31377.878} C_VEL
LIN {X 0,Y 687.321,Z 861.934,A -85,B 0,C 180,E1 31376.74,E2 31376.74} C_VEL
LIN {X 0,Y 688.435,Z 839.675,A -85,B 0,C 180,E1 31375.553,E2 31375.553} C_VEL
LIN {X 0,Y 689.517,Z 816.288,A -85,B 0,C 180,E1 31374.495,E2 31374.495} C_VEL
LIN {X 0,Y 690.364,Z 796.621,A -85,B 0,C 180,E1 31373.726,E2 31373.726} C_VEL
LIN {X 0,Y 691.221,Z 775.03,A -85,B 0,C 180,E1 31373.004,E2 31373.004} C_VEL
LIN {X 0,Y 692.057,Z 749.132,A -85,B 0,C 180,E1 31372.301,E2 31372.301} C_VEL
LIN {X 0,Y 692.629,Z 726.252,A -85,B 0,C 180,E1 31371.823,E2 31371.823} C_VEL
LIN {X 0,Y 693.116,Z 702.96,A -85,B 0,C 180,E1 31371.465,E2 31371.465} C_VEL
LIN {X 0,Y 695.381,Z 461.516,A -85,B 0,C 180,E1 31368.534,E2 31368.534} C_VEL
LIN {X 0,Y 696.836,Z 297.234,A -85,B 0,C 180,E1 31366.483,E2 31366.483} C_VEL
LIN {X 0,Y 694.778,Z 290.127,A -85,B 0,C 180,E1 31366.243,E2 31366.243} C_VEL
LIN {X 0,Y 687.074,Z 277.512,A -85,B 0,C 180,E1 31365.487,E2 31365.487} C_VEL
LIN {X 0,Y 681.332,Z 263.922,A -85,B 0,C 180,E1 31363.96,E2 31363.96} C_VEL
LIN {X 0,Y 680.479,Z 261.379,A -85,B 0,C 180,E1 31363.646,E2 31363.646} C_VEL
LIN {X 0,Y 680.455,Z 261.211,A -85,B 0,C 180,E1 31361.06,E2 31361.06} C_VEL
LIN {X 0,Y 680.508,Z 261.201,A -85,B 0,C 180,E1 31358.042,E2 31358.042} C_VEL
LIN {X 0,Y 680.448,Z 261.217,A -85,B 0,C 180,E1 31355.275,E2 31355.275} C_VEL
LIN {X 0,Y 680.493,Z 261.216,A -85,B 0,C 180,E1 31352.533,E2 31352.533} C_VEL
LIN {X 0,Y 680.463,Z 261.212,A -85,B 0,C 180,E1 31349.489,E2 31349.489} C_VEL
LIN {X 0,Y 680.453,Z 261.213,A -85,B 0,C 180,E1 31346.881,E2 31346.881} C_VEL
LIN {X 0,Y 680.524,Z 261.211,A -85,B 0,C 180,E1 31343.924,E2 31343.924} C_VEL
LIN {X 0,Y 680.448,Z 261.206,A -85,B 0,C 180,E1 31341.077,E2 31341.077} C_VEL
LIN {X 0,Y 680.488,Z 261.204,A -85,B 0,C 180,E1 31338.339,E2 31338.339} C_VEL
LIN {X 0,Y 680.461,Z 261.205,A -85,B 0,C 180,E1 31335.25,E2 31335.25} C_VEL
LIN {X 0,Y 680.451,Z 261.198,A -85,B 0,C 180,E1 31332.647,E2 31332.647} C_VEL
LIN {X 0,Y 680.518,Z 261.207,A -85,B 0,C 180,E1 31329.643,E2 31329.643} C_VEL
LIN {X 0,Y 680.446,Z 261.186,A -85,B 0,C 180,E1 31326.836,E2 31326.836} C_VEL
LIN {X 0,Y 680.485,Z 261.212,A -85,B 0,C 180,E1 31324.129,E2 31324.129} C_VEL
LIN {X 0,Y 680.46,Z 261.196,A -85,B 0,C 180,E1 31321.01,E2 31321.01} C_VEL
LIN {X 0,Y 680.454,Z 261.203,A -85,B 0,C 180,E1 31318.4,E2 31318.4} C_VEL
LIN {X 0,Y 680.522,Z 261.205,A -85,B 0,C 180,E1 31315.449,E2 31315.449} C_VEL
LIN {X 0,Y 680.446,Z 261.189,A -85,B 0,C 180,E1 31312.57,E2 31312.57} C_VEL
LIN {X 0,Y 680.493,Z 261.213,A -85,B 0,C 180,E1 31309.844,E2 31309.844} C_VEL
LIN {X 0,Y 680.458,Z 261.19,A -85,B 0,C 180,E1 31306.748,E2 31306.748} C_VEL
LIN {X 0,Y 680.455,Z 261.208,A -85,B 0,C 180,E1 31304.138,E2 31304.138} C_VEL
LIN {X 0,Y 680.513,Z 261.196,A -85,B 0,C 180,E1 31301.126,E2 31301.126} C_VEL
LIN {X 0,Y 680.449,Z 261.206,A -85,B 0,C 180,E1 31298.356,E2 31298.356} C_VEL
LIN {X 0,Y 680.489,Z 261.217,A -85,B 0,C 180,E1 31295.644,E2 31295.644} C_VEL
LIN {X 0,Y 680.465,Z 261.212,A -85,B 0,C 180,E1 31292.564,E2 31292.564} C_VEL
LIN {X 0,Y 680.457,Z 261.217,A -85,B 0,C 180,E1 31289.939,E2 31289.939} C_VEL
LIN {X 0,Y 680.519,Z 261.184,A -85,B 0,C 180,E1 31286.967,E2 31286.967} C_VEL
LIN {X 0,Y 680.452,Z 261.217,A -85,B 0,C 180,E1 31284.104,E2 31284.104} C_VEL
LIN {X 0,Y 680.494,Z 261.187,A -85,B 0,C 180,E1 31281.356,E2 31281.356} C_VEL
LIN {X 0,Y 680.462,Z 261.214,A -85,B 0,C 180,E1 31278.285,E2 31278.285} C_VEL
LIN {X 0,Y 680.461,Z 261.22,A -85,B 0,C 180,E1 31275.617,E2 31275.617} C_VEL
LIN {X 0,Y 680.481,Z 261.422,A -85,B 0,C 180,E1 31274.028,E2 31274.028} C_VEL
LIN {X 0,Y 688.286,Z 280.065,A -85,B 0,C 180,E1 31271.932,E2 31271.932} C_VEL
